    ELSIF (_eJobReslt = E_PROGRESS.PROGRESS_DONE)
    THEN
      _eState                   := E_PROGRESS.PROGRESS_CHECK;
      _eJobReslt                := _GroupItf.Enable(FALSE);
    END_IF
END_CASE
//-----------------------------------------------------------------------------
//-----------------------------------------------------------------------------
CASE _eState
OF
  E_PROGRESS.PROGRESS_CHECK:
    IF (_GroupInfo.GroupStandby) OR
       (_GroupInfo.GroupMoving)  OR
       (_GroupInfo.GroupNotReady)
    THEN
      _eState                   := E_PROGRESS.PROGRESS_DONE;

      IF (_eMessageLevel = E_MessageType.eMessageVerbose)
      THEN
        _stMsg.eType            := E_MessageType.eMessageVerbose;
        _stMsg.eSubdevice       := e_Subdevice.TransportUnit_General;
        _stMsg.iErrorNumber     := 0;
        _stMsg.sText            := concat( 'State: ', TO_STRING(THIS^._eState));
        _stMsg.sText            := concat(_stMsg.sText, ': ');
        _stMsg.sText            := concat(_stMsg.sText, TO_STRING(_eState));
        f_MessageSet(_stMsg, _nXpu);
      END_IF
    ELSE
      IF (_GroupInfo.GroupErrorStop) OR
         (_GroupInfo.GroupError)
      THEN
        _eState                 := E_PROGRESS.PROGRESS_ERROR;
      END_IF
    END_IF
END_CASE
//-----------------------------------------------------------------------------
//-----------------------------------------------------------------------------
GroupEnable                     := _eState;
END_METHOD

PROPERTY GroupInfo : REFERENCE TO ST_GROUP_INFO
SET
_GroupInfo REF= GroupInfo;
END_SET
END_PROPERTY

PROPERTY GroupItf : I_XtsTransport_CaGroup
SET
_GroupItf := GroupItf;
END_SET
END_PROPERTY

METHOD GroupStop : E_PROGRESS
VAR_INPUT
  Execute     : BOOL;
END_VAR
VAR_INST
  _nRepeat,
  _nStation,
  _nErrorId   : UDINT;
  _eJobReslt,
  _eState     : E_PROGRESS;
END_VAR
//-----------------------------------------------------------------------------
IF NOT Execute 
THEN 
	_eState                      := E_PROGRESS.PROGRESS_INIT; 
END_IF 
//-----------------------------------------------------------------------------
IF NOT Check() 
THEN 
	GroupStop                    := E_PROGRESS.PROGRESS_ERROR; 
	RETURN; 
END_IF
//-----------------------------------------------------------------------------
//-----------------------------------------------------------------------------
CASE _eState
OF
  E_PROGRESS.PROGRESS_INIT:
    IF Execute
    THEN
      _nRepeat                  :=
      _nErrorId                 := 0;
      _eJobReslt                := _GroupItf.Stop(FALSE);

      _eState                   := E_PROGRESS.PROGRESS_BUSY;
    END_IF
END_CASE
//---------------------------------------------------------------------------
//---------------------------------------------------------------------------
CASE _eState
OF
  E_PROGRESS.PROGRESS_BUSY:
    _eJobReslt                  := _GroupItf.Stop(TRUE);

    IF (_eJobReslt = E_PROGRESS.PROGRESS_ERROR)
    THEN
      _eState                   := E_PROGRESS.PROGRESS_PREPARE;
      _nErrorId                 := _GroupInfo.GroupErrorId;
      _eJobReslt                := _GroupItf.Stop(FALSE);

    ELSIF (_eJobReslt = E_PROGRESS.PROGRESS_DONE)
    THEN
      _eState                   := E_PROGRESS.PROGRESS_WORKING;
      _eJobReslt                := _GroupItf.Stop(FALSE);
    END_IF
END_CASE
//-----------------------------------------------------------------------------
//-----------------------------------------------------------------------------
CASE _eState
OF
  E_PROGRESS.PROGRESS_WORKING:
    IF NOT (_GroupInfo.GroupError)
    THEN
      _eState                   := E_PROGRESS.PROGRESS_DONE;

      IF (_eMessageLevel = E_MessageType.eMessageVerbose)
      THEN
        _stMsg.eType            := E_MessageType.eMessageVerbose;
        _stMsg.eSubdevice       := e_Subdevice.TransportUnit_General;
        _stMsg.iErrorNumber     := 0;
        _stMsg.sText            := concat( 'State: ', TO_STRING(THIS^._eState));
        _stMsg.sText            := concat(_stMsg.sText, ': ');
        _stMsg.sText            := concat(_stMsg.sText, TO_STRING(_eState));
        f_MessageSet(_stMsg, _nXpu);
      END_IF
    ELSE
      IF (_GroupInfo.GroupErrorStop) OR
         (_GroupInfo.GroupError)
      THEN
        _nRepeat                := _nRepeat + 1;
        IF NOT (_nRepeat > 2)
        THEN
          _eState               := E_PROGRESS.PROGRESS_BUSY;
        ELSE
          _eState               := E_PROGRESS.PROGRESS_ERROR;
        END_IF
      END_IF
    END_IF
END_CASE
//-----------------------------------------------------------------------------
//-----------------------------------------------------------------------------

GroupStop                       := _eState;
END_METHOD

PROPERTY MessageLevel : e_messagetype
SET
_eMessageLevel := MessageLevel;
END_SET
END_PROPERTY

METHOD MoverDisableAll : e_progress
VAR_INPUT
  Execute     : BOOL;
END_VAR
VAR_INST
  _nMover     : UINT;
  _nErrorId   : UDINT;
  _eRslt,
  _eState     : E_PROGRESS;
END_VAR
//-----------------------------------------------------------------------------
IF NOT Execute 
THEN 
	_eState                       := E_PROGRESS.PROGRESS_INIT; 
END_IF 
//-----------------------------------------------------------------------------
IF NOT Check() 
THEN 
	MoverDisableAll               := E_PROGRESS.PROGRESS_ERROR; 
	RETURN; 
END_IF
//-----------------------------------------------------------------------------
//-----------------------------------------------------------------------------
CASE _eState
OF
  E_PROGRESS.PROGRESS_INIT:
    IF Execute
    THEN
      _nErrorId                 := 0;
      _nMover                   := 1;

      _eState                   := E_PROGRESS.PROGRESS_BUSY;
    END_IF
END_CASE
//-----------------------------------------------------------------------------
//-----------------------------------------------------------------------------
CASE _eState
OF
  E_PROGRESS.PROGRESS_BUSY:
    _eState                     := E_PROGRESS.PROGRESS_PREPARE;
    _eRslt                      := _MoverItf[_nMover].Disable(FALSE);
    _eRslt                      := _MoverItf[_nMover].Reset(FALSE);
END_CASE
//-----------------------------------------------------------------------------
//-----------------------------------------------------------------------------
CASE _eState
OF
  E_PROGRESS.PROGRESS_PREPARE:
    _eRslt                      := _MoverItf[_nMover].Disable(TRUE);

    IF (_eRslt = E_PROGRESS.PROGRESS_ERROR)
    THEN
      _eState                   := E_PROGRESS.PROGRESS_BUSY;
      _nErrorId                 := _MoverInfo[_nMover].nErrorId; 
      _eRslt                    := _MoverItf[_nMover].Disable(FALSE);
      _MoverItf[_nMover].Reset(TRUE);

    ELSIF (_eRslt = E_PROGRESS.PROGRESS_DONE)
    THEN
      _eState                   := E_PROGRESS.PROGRESS_STARTUP;
    END_IF
END_CASE
//-----------------------------------------------------------------------------
//-----------------------------------------------------------------------------
CASE _eState
OF
  E_PROGRESS.PROGRESS_STARTUP:
    _eState                     := E_PROGRESS.PROGRESS_CHECK;
    _eRslt                      := _MoverItf[_nMover].Disable(FALSE);
END_CASE
//-----------------------------------------------------------------------------
//-----------------------------------------------------------------------------
CASE _eState
OF
  E_PROGRESS.PROGRESS_CHECK:
    IF (_nMover > MAX_MOVER-1)
    THEN
      _eState                   := E_PROGRESS.PROGRESS_DONE;

      IF (_eMessageLevel = E_MessageType.eMessageVerbose)
      THEN
        _stMsg.eType            := E_MessageType.eMessageVerbose;
        _stMsg.eSubdevice       := e_Subdevice.TransportUnit_General;
        _stMsg.iErrorNumber     := 0;
        _stMsg.sText            := concat( 'State: ', TO_STRING(THIS^._eState));
        _stMsg.sText            := concat(_stMsg.sText, ': ');
        _stMsg.sText            := concat(_stMsg.sText, TO_STRING(_eState));
        f_MessageSet(_stMsg, _nXpu);
      END_IF
    ELSE
      _nMover                   := _nMover + 1;
      _eState                   := E_PROGRESS.PROGRESS_BUSY;
    END_IF
END_CASE
//-----------------------------------------------------------------------------
//-----------------------------------------------------------------------------

MoverDisableAll                 := _eState;
END_METHOD

METHOD MoverEnableAll : e_progress
VAR_INPUT
  Execute     : BOOL;
END_VAR
VAR_INST
  _nMover     : UINT;
  _nErrorId   : UDINT;
  _eRslt,
  _eState     : E_PROGRESS;
END_VAR
//-----------------------------------------------------------------------------
IF NOT Execute 
THEN 
	_eState                       := E_PROGRESS.PROGRESS_INIT; 
END_IF 
//-----------------------------------------------------------------------------
IF NOT Check() 
THEN 
	MoverEnableAll                := E_PROGRESS.PROGRESS_ERROR; 
	RETURN; 
END_IF
//-----------------------------------------------------------------------------
//-----------------------------------------------------------------------------
CASE _eState
OF
  E_PROGRESS.PROGRESS_INIT:
    IF Execute
    THEN
      _nErrorId                 := 0;
      _nMover                   := 1;

      _eState                   := E_PROGRESS.PROGRESS_BUSY;
    END_IF
END_CASE
//-----------------------------------------------------------------------------
//-----------------------------------------------------------------------------
CASE _eState
OF
  E_PROGRESS.PROGRESS_BUSY:
    _eState                     := E_PROGRESS.PROGRESS_PREPARE;
    _eRslt                      := _MoverItf[_nMover].Enable(FALSE);
    _eRslt                      := _MoverItf[_nMover].Reset (FALSE);
END_CASE
//-----------------------------------------------------------------------------
//-----------------------------------------------------------------------------
CASE _eState
OF
  E_PROGRESS.PROGRESS_PREPARE:
    _eRslt                      := _MoverItf[_nMover].Enable(TRUE);

    IF (_eRslt = E_PROGRESS.PROGRESS_ERROR)
    THEN
      _eState                   := E_PROGRESS.PROGRESS_BUSY;
      _nErrorId                 := _MoverInfo[_nMover].nErrorId;
      _MoverItf[_nMover].Reset (TRUE);

    ELSIF (_eRslt = E_PROGRESS.PROGRESS_DONE)
    THEN
      _eState                   := E_PROGRESS.PROGRESS_STARTUP;
    END_IF
END_CASE
//-----------------------------------------------------------------------------
//-----------------------------------------------------------------------------
CASE _eState
OF
  E_PROGRESS.PROGRESS_STARTUP:
    _eState                     := E_PROGRESS.PROGRESS_CHECK;
    _eRslt                      := _MoverItf[_nMover].Enable(FALSE);
END_CASE
//-----------------------------------------------------------------------------
//-----------------------------------------------------------------------------
CASE _eState
OF
  E_PROGRESS.PROGRESS_CHECK:
    IF (_nMover > MAX_MOVER-1)
    THEN
      _eState                   := E_PROGRESS.PROGRESS_DONE;
      IF (_eMessageLevel = E_MessageType.eMessageVerbose)
      THEN
        _stMsg.eType            := E_MessageType.eMessageVerbose;
        _stMsg.eSubdevice       := e_Subdevice.TransportUnit_General;
        _stMsg.iErrorNumber     := 0;
        _stMsg.sText            := concat( 'State: ', TO_STRING(THIS^._eState));
        _stMsg.sText            := concat(_stMsg.sText, ': ');
        _stMsg.sText            := concat(_stMsg.sText, TO_STRING(_eState));
        f_MessageSet(_stMsg, _nXpu);
      END_IF
    ELSE
      _nMover                   := _nMover + 1;
      _eState                   := E_PROGRESS.PROGRESS_BUSY;
    END_IF
END_CASE
//-----------------------------------------------------------------------------
//-----------------------------------------------------------------------------

MoverEnableAll                  := _eState;
END_METHOD

METHOD MoverHaltAll : e_progress
VAR_INPUT
  Execute     : BOOL;
END_VAR
VAR_INST
  _nMover     : UINT;
  _nErrorId   : UDINT;
  _eRslt,
  _eState     : E_PROGRESS;
  _stMoveData : ST_MOVE_DATA; // dyn constraints for _MoverItf[i].Halt(Execute, stMoveData)
END_VAR
//-----------------------------------------------------------------------------
IF NOT Execute 
THEN 
	_eState                       := E_PROGRESS.PROGRESS_INIT; 
END_IF 
//-----------------------------------------------------------------------------
IF NOT Check() 
THEN 
	MoverHaltAll                  := E_PROGRESS.PROGRESS_ERROR; 
	RETURN; 
END_IF
//-----------------------------------------------------------------------------
//-----------------------------------------------------------------------------
CASE _eState
OF
  E_PROGRESS.PROGRESS_INIT:
    IF Execute
    THEN
      _nErrorId                 := 0;
      _nMover                   := 1;

      _eState                   := E_PROGRESS.PROGRESS_BUSY;
    END_IF
END_CASE
//-----------------------------------------------------------------------------
//-----------------------------------------------------------------------------
CASE _eState
OF
  E_PROGRESS.PROGRESS_BUSY:
    _eState                     := E_PROGRESS.PROGRESS_PREPARE;
    _stMoveData.rAcc            := _StationStart.rAccDec;
    _stMoveData.rGap            := _MoverLastGap[_nMover];

    IF NOT (_GroupInfo.AxisCount = MAX_MOVER)
    THEN
      _eRslt                    := _MoverItf[_nMover].Halt(FALSE, _stMoveData);
    ELSE
      _eRslt                    := _MoverItf[_nMover].HaltCa(FALSE, _stMoveData);
    END_IF
END_CASE
//-----------------------------------------------------------------------------
//-----------------------------------------------------------------------------
CASE _eState
OF
  E_PROGRESS.PROGRESS_PREPARE:
    IF NOT (_GroupInfo.AxisCount = MAX_MOVER)
    THEN
      _eRslt                    := _MoverItf[_nMover].Halt(TRUE, _stMoveData);
    ELSE
      _eRslt                    := _MoverItf[_nMover].HaltCa(TRUE, _stMoveData);
    END_IF

    IF (_eRslt = E_PROGRESS.PROGRESS_ERROR)
    THEN
      _eState                   := E_PROGRESS.PROGRESS_WORKING; // reset error on purpose, since we have to come back and get everybody in standstill
      _eRslt                    := _MoverItf[_nMover].Reset(FALSE);
      _nErrorId                 := _MoverInfo[_nMover].nErrorId; 

    ELSIF (_eRslt = E_PROGRESS.PROGRESS_DONE)
    THEN
      _eState                   := E_PROGRESS.PROGRESS_STARTUP;
    END_IF
END_CASE
//-----------------------------------------------------------------------------
//-----------------------------------------------------------------------------
CASE _eState
OF
  E_PROGRESS.PROGRESS_STARTUP:
    _eState                     := E_PROGRESS.PROGRESS_CHECK;

    IF NOT (_GroupInfo.AxisCount = MAX_MOVER)
    THEN
      _eRslt                    := _MoverItf[_nMover].Halt(FALSE, _stMoveData);
    ELSE
      _eRslt                    := _MoverItf[_nMover].HaltCa(FALSE, _stMoveData);
    END_IF

END_CASE
//-----------------------------------------------------------------------------
//-----------------------------------------------------------------------------
CASE _eState
OF
  E_PROGRESS.PROGRESS_CHECK:
    IF (_nMover > MAX_MOVER-1)
    THEN
      _eState                   := E_PROGRESS.PROGRESS_OCCUPIED;
    ELSE
      _nMover                   := _nMover + 1;
      _eState                   := E_PROGRESS.PROGRESS_BUSY;
    END_IF
END_CASE
//-----------------------------------------------------------------------------
//-----------------------------------------------------------------------------
CASE _eState
OF
  E_PROGRESS.PROGRESS_OCCUPIED:
    IF (_GroupInfo.AllAxesStanding)
    THEN
      _eState                   := E_PROGRESS.PROGRESS_DONE;

      IF (_eMessageLevel = E_MessageType.eMessageVerbose)
      THEN
        _stMsg.eType            := E_MessageType.eMessageVerbose;
        _stMsg.eSubdevice       := e_Subdevice.TransportUnit_General;
        _stMsg.iErrorNumber     := 0;
        _stMsg.sText            := concat( 'State: ', TO_STRING(THIS^._eState));
        _stMsg.sText            := concat(_stMsg.sText, ': ');
        _stMsg.sText            := concat(_stMsg.sText, TO_STRING(_eState));
        f_MessageSet(_stMsg, _nXpu);
      END_IF
    ELSE
      _nMover                   := 1;
      _eState                   := E_PROGRESS.PROGRESS_BUSY;
    END_IF
END_CASE
//-----------------------------------------------------------------------------
//-----------------------------------------------------------------------------
CASE _eState
OF
  E_PROGRESS.PROGRESS_WORKING:
    _eRslt                      := _MoverItf[_nMover].Reset(TRUE);

    IF (_eRslt = E_PROGRESS.PROGRESS_ERROR)
    THEN
      _eRslt                    := _MoverItf[_nMover].Reset(FALSE);
      _nErrorId                 := _MoverInfo[_nMover].nErrorId; 

    ELSIF (_eRslt = E_PROGRESS.PROGRESS_DONE)
    THEN
      _eState                   := E_PROGRESS.PROGRESS_BUSY;
      _eRslt                    := _MoverItf[_nMover].Reset(FALSE);
    END_IF
END_CASE
//-----------------------------------------------------------------------------
//-----------------------------------------------------------------------------

MoverHaltAll                    := _eState;
END_METHOD

PROPERTY MoverInfo : REFERENCE TO ARRAY[1..MAX_MOVER] OF ST_MOVER_INFO
SET
_MoverInfo REF= MoverInfo;
END_SET
END_PROPERTY

PROPERTY MoverItf : reference TO ARRAY[1..MAX_MOVER] OF I_XtsTransport_Mover
SET
_MoverItf REF= MoverItf;
END_SET
END_PROPERTY

PROPERTY MoverLastGap : REFERENCE to ARRAY[1..MAX_MOVER] of LREAL
SET
_MoverLastGap REF= MoverLastGap;
END_SET
END_PROPERTY

PROPERTY MoverLastPosition : REFERENCE to ARRAY[1..MAX_MOVER] of LREAL
SET
_MoverLastPosition REF= MoverLastPosition;
END_SET
END_PROPERTY

METHOD MoverStopAll : e_progress
VAR_INPUT
  Execute     : BOOL;
END_VAR
VAR_INST
  _nMover     : UINT;
  _nErrorId   : UDINT;
  _eRslt,
  _eState     : E_PROGRESS;
  _stMoveData : ST_MOVE_DATA; // dyn constraints for _MoverItf[i].Halt(Execute, stMoveData)
END_VAR
//-----------------------------------------------------------------------------
IF NOT Execute 
THEN 
	_eState                       := E_PROGRESS.PROGRESS_INIT; 
END_IF 
//-----------------------------------------------------------------------------
IF NOT Check() 
THEN 
	MoverStopAll                  := E_PROGRESS.PROGRESS_ERROR; 
	RETURN; 
END_IF
//-----------------------------------------------------------------------------
//-----------------------------------------------------------------------------
CASE _eState
OF
  E_PROGRESS.PROGRESS_INIT:
    IF Execute
    THEN
      _nErrorId                 := 0;
      _nMover                   := 1;

      _eState                   := E_PROGRESS.PROGRESS_BUSY;
    END_IF
END_CASE
//-----------------------------------------------------------------------------
//-----------------------------------------------------------------------------
CASE _eState
OF
  E_PROGRESS.PROGRESS_BUSY:
    _eState                     := E_PROGRESS.PROGRESS_PREPARE;
    _stMoveData.rAcc            := _StationStart.rAccDec;
    _stMoveData.rGap            := _MoverLastGap[_nMover];

    _eRslt                      := _MoverItf[_nMover].Stop(FALSE, _stMoveData);
END_CASE
//-----------------------------------------------------------------------------
//-----------------------------------------------------------------------------
CASE _eState
OF
  E_PROGRESS.PROGRESS_PREPARE:
    _eRslt                      := _MoverItf[_nMover].Stop(TRUE, _stMoveData);

    IF (_eRslt = E_PROGRESS.PROGRESS_ERROR)
    THEN
      _eState                   := E_PROGRESS.PROGRESS_WORKING; // reset error on purpose, since we have to come back and get everybody in standstill
      _eRslt                    := _MoverItf[_nMover].Reset(FALSE);
      _nErrorId                 := _MoverInfo[_nMover].nErrorId; 

    ELSIF (_eRslt = E_PROGRESS.PROGRESS_DONE)
    THEN
      _eState                   := E_PROGRESS.PROGRESS_STARTUP;
    END_IF
END_CASE
//-----------------------------------------------------------------------------
//-----------------------------------------------------------------------------
CASE _eState
OF
  E_PROGRESS.PROGRESS_STARTUP:
    _eState                     := E_PROGRESS.PROGRESS_CHECK;
    _eRslt                      := _MoverItf[_nMover].Halt(FALSE, _stMoveData);
END_CASE
//-----------------------------------------------------------------------------
//-----------------------------------------------------------------------------
CASE _eState
OF
  E_PROGRESS.PROGRESS_CHECK:
    IF (_nMover > MAX_MOVER-1)
    THEN
      _eState                   := E_PROGRESS.PROGRESS_OCCUPIED;
    ELSE
      _nMover                   := _nMover + 1;
      _eState                   := E_PROGRESS.PROGRESS_BUSY;
    END_IF
END_CASE
//-----------------------------------------------------------------------------
//-----------------------------------------------------------------------------
CASE _eState
OF
  E_PROGRESS.PROGRESS_OCCUPIED:
    IF (_GroupInfo.AllAxesStanding)
    THEN
      _eState                   := E_PROGRESS.PROGRESS_DONE;

      IF (_eMessageLevel = E_MessageType.eMessageVerbose)
      THEN
        _stMsg.eType            := E_MessageType.eMessageVerbose;
        _stMsg.eSubdevice       := e_Subdevice.TransportUnit_General;
        _stMsg.iErrorNumber     := 0;
        _stMsg.sText            := concat( 'State: ', TO_STRING(THIS^._eState));
        _stMsg.sText            := concat(_stMsg.sText, ': ');
        _stMsg.sText            := concat(_stMsg.sText, TO_STRING(_eState));
        f_MessageSet(_stMsg, _nXpu);
      END_IF
    ELSE
      _nMover                   := 1;
      _eState                   := E_PROGRESS.PROGRESS_BUSY;
    END_IF
END_CASE
//-----------------------------------------------------------------------------
//-----------------------------------------------------------------------------
CASE _eState
OF
  E_PROGRESS.PROGRESS_WORKING:
    _eRslt                      := _MoverItf[_nMover].Reset(TRUE);

    IF (_eRslt = E_PROGRESS.PROGRESS_ERROR)
    THEN
      _eRslt                    := _MoverItf[_nMover].Reset(FALSE);
      _nErrorId                 := _MoverInfo[_nMover].nErrorId; 

    ELSIF (_eRslt = E_PROGRESS.PROGRESS_DONE)
    THEN
      _eState                   := E_PROGRESS.PROGRESS_BUSY;
      _eRslt                    := _MoverItf[_nMover].Reset(FALSE);
    END_IF
END_CASE
//-----------------------------------------------------------------------------
//-----------------------------------------------------------------------------

MoverStopAll                    := _eState;
END_METHOD

PROPERTY State : REFERENCE TO ST_XTS_TRANSPORT_STATE
SET
_State ref= State;
END_SET
END_PROPERTY

PROPERTY StationControl : REFERENCE TO ARRAY[1..MAX_STATION]  OF ST_STATION_CTRL
SET
_StationControl REF= StationControl;
END_SET
END_PROPERTY

PROPERTY StationCtrlItf : REFERENCE TO ARRAY[1..MAX_STATION]  OF I_XtsTransport_Station;
SET
_ItfStationCtrl REF= StationCtrlItf;
END_SET
END_PROPERTY

PROPERTY StationListsItf : reference to ARRAY[1..MAX_STATION] OF I_Station_LinkedList
SET
_ItfStationList ref= StationListsItf;
END_SET
END_PROPERTY

METHOD StationsClearAll : E_PROGRESS
VAR_INPUT
  Execute     : BOOL;
END_VAR
VAR_INST
  _nStation,
  _nErrorId   : UDINT;
  _eJobReslt,
  _eState     : E_PROGRESS;
END_VAR
//-----------------------------------------------------------------------------
IF NOT Execute 
THEN 
	_eState                       := E_PROGRESS.PROGRESS_INIT; 
END_IF 
//-----------------------------------------------------------------------------
IF NOT Check() 
THEN 
	StationsClearAll              := E_PROGRESS.PROGRESS_ERROR; 
	RETURN; 
END_IF
//-----------------------------------------------------------------------------
//-----------------------------------------------------------------------------
CASE _eState
OF
  E_PROGRESS.PROGRESS_INIT:
    IF Execute
    THEN
      _nErrorId                 := 0;
      _nStation                 := 1;
      _eState                   := E_PROGRESS.PROGRESS_BUSY;
    END_IF
  //---------------------------------------------------------------------------
  //---------------------------------------------------------------------------
  E_PROGRESS.PROGRESS_BUSY:
    _eJobReslt                  := _ItfStationCtrl[_nStation].Init();

    IF (_eJobReslt = E_PROGRESS.PROGRESS_ERROR)
    THEN
      _eState                   := E_PROGRESS.PROGRESS_ERROR;
      _nErrorId                 := 669;

    ELSIF (_eJobReslt = E_PROGRESS.PROGRESS_DONE)
    THEN
      _eState                   := E_PROGRESS.PROGRESS_WORKING;
    END_IF

  //---------------------------------------------------------------------------
  //---------------------------------------------------------------------------
  E_PROGRESS.PROGRESS_WORKING:
    IF (_nStation < MAX_STATION)
    THEN
      _nStation                 := _nStation + 1;
      _eState                   := E_PROGRESS.PROGRESS_BUSY;
    ELSE
      _eState                   := E_PROGRESS.PROGRESS_DONE;

      IF (_eMessageLevel = E_MessageType.eMessageVerbose)
      THEN
        _stMsg.eType            := E_MessageType.eMessageVerbose;
        _stMsg.eSubdevice       := e_Subdevice.TransportUnit_General;
        _stMsg.iErrorNumber     := 0;
        _stMsg.sText            := concat( 'State: ', TO_STRING(THIS^._eState));
        _stMsg.sText            := concat(_stMsg.sText, ': ');
        _stMsg.sText            := concat(_stMsg.sText, TO_STRING(_eState));
        f_MessageSet(_stMsg, _nXpu);
      END_IF
    END_IF
END_CASE
//-----------------------------------------------------------------------------
//-----------------------------------------------------------------------------

StationsClearAll                := _eState;
END_METHOD

METHOD StationsClearOutfeed : e_progress
VAR_INPUT
  Execute         : BOOL;
END_VAR
VAR_INST
  _StnState       : ST_STATION_STATE;

  _nStation,
  _nMover         : UINT;

  _nErrorId       : UDINT;

  _eRslt,
  _eState         : E_PROGRESS;
  
  _stMsg          : ST_Message;
  _stMoveData     : ST_MOVE_DATA;
END_VAR
//-----------------------------------------------------------------------------
IF NOT Execute 
THEN 
	_eState                       := E_PROGRESS.PROGRESS_INIT; 
END_IF 
//-----------------------------------------------------------------------------
IF NOT Check() 
THEN 
	StationsClearOutfeed           := E_PROGRESS.PROGRESS_ERROR; 
	RETURN; 
END_IF
//-----------------------------------------------------------------------------
//-----------------------------------------------------------------------------
CASE _eState
OF
  E_PROGRESS.PROGRESS_INIT:
    IF Execute
    THEN
      _nErrorId                 := 0;

      _nStation                 :=
      _nMover                   := 1;

      _eState                   := E_PROGRESS.PROGRESS_BUSY;
    END_IF
END_CASE
//-----------------------------------------------------------------------------
//-----------------------------------------------------------------------------
CASE _eState
OF
  E_PROGRESS.PROGRESS_BUSY:
    _StnState                   := _StationState[_nStation];

    CASE _StnState.eState
    OF
      E_STATION_STATE.STATION_MOVER_RELEASE:
        _StationControl[_nStation].eCmd := E_STATION_CTRL.STATION_MOVER_GONE;

    ELSE
      _eState                   := E_PROGRESS.PROGRESS_PREPARE;  
    END_CASE
END_CASE
//-----------------------------------------------------------------------------
//-----------------------------------------------------------------------------
CASE _eState
OF
  E_PROGRESS.PROGRESS_PREPARE:
    IF (_nStation > MAX_STATION-1)
    THEN
      _eState                   := E_PROGRESS.PROGRESS_DONE;
    ELSE
      _nStation                 := _nStation + 1;
      _eState                   := E_PROGRESS.PROGRESS_BUSY;
    END_IF
END_CASE

StationsClearOutfeed             := _eState;
END_METHOD

PROPERTY StationStart : reference to ST_STATION_PARAMETER
SET
_StationStart REF= StationStart;
END_SET
END_PROPERTY

PROPERTY StationStartIndex : uint
GET
StationStartIndex := _nStartStation;
END_GET
SET
_nStartStation := StationStartIndex;
END_SET
END_PROPERTY

PROPERTY StationState : REFERENCE TO ARRAY[1..MAX_STATION]  OF ST_STATION_STATE
SET
_StationState REF= StationState;
END_SET
END_PROPERTY

METHOD Template : E_PROGRESS
VAR_INPUT
  Execute     : BOOL;
END_VAR
VAR_INST
  _nErrorId   : UDINT;
  _eState     : E_PROGRESS;
END_VAR
//-----------------------------------------------------------------------------
IF NOT Execute 
THEN 
	_eState                       := E_PROGRESS.PROGRESS_INIT; 
END_IF 
//-----------------------------------------------------------------------------
IF NOT Check() 
THEN 
	Template_1                    := E_PROGRESS.PROGRESS_ERROR; 
	RETURN; 
END_IF
//-----------------------------------------------------------------------------
//-----------------------------------------------------------------------------
CASE _eState
OF
  E_PROGRESS.PROGRESS_INIT:
    IF Execute
    THEN
      _nErrorId                 := 0;

      _eState                   := E_PROGRESS.PROGRESS_BUSY;
    END_IF
END_CASE
//-----------------------------------------------------------------------------
//-----------------------------------------------------------------------------
CASE _eState
OF
  E_PROGRESS.PROGRESS_BUSY:
    _eState                     := E_PROGRESS.PROGRESS_PREPARE;
END_CASE
//-----------------------------------------------------------------------------
//-----------------------------------------------------------------------------
CASE _eState
OF
  E_PROGRESS.PROGRESS_PREPARE:

    IF (.Error)
    THEN
      _eState                   := E_PROGRESS.PROGRESS_ERROR;
      _nErrorId                 := 


    ELSIF (.Done)
    THEN
      _eState                   := E_PROGRESS.;

    END_IF
END_CASE
//-----------------------------------------------------------------------------
//-----------------------------------------------------------------------------

Template_1                      := _eState;
END_METHOD

METHOD TransportRestart : e_progress // movers must already to be error free, enabled and added to CA Group
VAR_INPUT
  Execute         : BOOL;
END_VAR
VAR_INST
  _StnState       : ST_STATION_STATE;

  _nStation,
  _nMover         : UINT;

  _nErrorId       : UDINT;

  _eRslt,
  _eState         : E_PROGRESS;
  
  _stMsg          : ST_Message;
  _stMoveData     : ST_MOVE_DATA;
END_VAR
//-----------------------------------------------------------------------------
IF NOT Execute 
THEN 
	_eState                       := E_PROGRESS.PROGRESS_INIT; 
END_IF 
//-----------------------------------------------------------------------------
IF NOT Check() 
THEN 
	TransportRestart              := E_PROGRESS.PROGRESS_ERROR; 
	RETURN; 
END_IF
//-----------------------------------------------------------------------------
//-----------------------------------------------------------------------------
CASE _eState
OF
  E_PROGRESS.PROGRESS_INIT:
    IF Execute
    THEN
      _nErrorId                 := 0;

      _nStation                 :=
      _nMover                   := 1;

      IF (_GroupInfo.AxisCountEnabled = MAX_MOVER)
      THEN
        _eState                 := E_PROGRESS.PROGRESS_BUSY;
      ELSE
        _eState                 := E_PROGRESS.PROGRESS_ERROR;

        _stMsg.eType            := E_MessageType.eMessageError;
        _stMsg.eSubdevice       := e_Subdevice.TransportUnit_Restart;
        _stMsg.iErrorNumber     := _GroupInfo.AxisCountEnabled;
        _stMsg.sText            := TO_STRING(_eState);
        _stMsg.sText            := concat(_stMsg.sText, ': _GroupInfo.AxisCountEnabled <> MAX_MOVER');
        f_MessageSet(_stMsg, _nXpu);
      END_IF
    END_IF
END_CASE
//-----------------------------------------------------------------------------
//-----------------------------------------------------------------------------
CASE _eState
OF
  E_PROGRESS.PROGRESS_BUSY:
    _StnState                   := _StationState[_nStation];

    CASE _StnState.eState
    OF
      E_STATION_STATE.STATION_ERROR_INFEED_ERROR:
        _StationControl[_nStation].eCmd := E_STATION_CTRL.STATION_MOVER_ENTER_RETRY;

      E_STATION_STATE.STATION_ERROR_OUTFEED_ERROR:
        _StationControl[_nStation].eCmd := E_STATION_CTRL.STATION_MOVER_GONE;

      E_STATION_STATE.STATION_ERROR_FATAL:
        _eState                 := E_PROGRESS.PROGRESS_ERROR;

        _stMsg.eType            := E_MessageType.eMessageError;
        _stMsg.eSubdevice       := e_Subdevice.TransportUnit_Restart;
        _stMsg.iErrorNumber     := _nStation;
        _stMsg.sText            := TO_STRING(_eState);
        _stMsg.sText            := concat(_stMsg.sText, ': _nStation STATION_ERROR_FATAL');
        f_MessageSet(_stMsg, _nXpu);

    ELSE
      _eState                   := E_PROGRESS.PROGRESS_PREPARE;  
    END_CASE
END_CASE
//-----------------------------------------------------------------------------
//-----------------------------------------------------------------------------
CASE _eState
OF
  E_PROGRESS.PROGRESS_PREPARE:
    IF (_nStation > MAX_STATION-1)
    THEN
      _eState                   := E_PROGRESS.PROGRESS_STARTUP;
    ELSE
      _nStation                 := _nStation + 1;
      _eState                   := E_PROGRESS.PROGRESS_BUSY;
    END_IF
END_CASE
//-----------------------------------------------------------------------------
//-----------------------------------------------------------------------------
CASE _eState
OF
  E_PROGRESS.PROGRESS_STARTUP:
    _stMoveData.rPos            := _MoverLastPosition[_nMover];
    _stMoveData.rGap            := _MoverLastGap     [_nMover];

    _stMoveData.rVelo           := _StationStart.rVelo;
    _stMoveData.rAcc            := _StationStart.rAccDec;
    _stMoveData.rJerk           := _StationStart.rJerk;

    _stMoveData.rDelta          :=   0.1;
    _stMoveData.rDistance       :=  -1.0;
    _stMoveData.rOverride       := 100.0;

    _eRslt                      := _MoverItf[_nMover].SendToAbsPosCa(FALSE, _stMoveData);

    IF (_MoverInfo[_nMover].bMoverEnabled)
    THEN
      _eState                   := E_PROGRESS.PROGRESS_CHECK;
    END_IF
END_CASE
//-----------------------------------------------------------------------------
//-----------------------------------------------------------------------------
CASE _eState
OF
  E_PROGRESS.PROGRESS_CHECK:
    _eRslt                      := _MoverItf[_nMover].SendToAbsPosCa(TRUE, _stMoveData);

    IF (_eRslt = E_PROGRESS.PROGRESS_ERROR)
    THEN
      _eState                   := E_PROGRESS.PROGRESS_ERROR;

    ELSIF (_eRslt = E_PROGRESS.PROGRESS_DONE)
    THEN
      _eRslt                    := _MoverItf[_nMover].SendToAbsPosCa(FALSE, _stMoveData);
      _eState                   := E_PROGRESS.PROGRESS_OCCUPIED;
    END_IF
END_CASE
//-----------------------------------------------------------------------------
//-----------------------------------------------------------------------------
CASE _eState
OF
  E_PROGRESS.PROGRESS_OCCUPIED:
    IF (_nMover > MAX_MOVER-1)
    THEN
      _eState                   := E_PROGRESS.PROGRESS_DONE;

      IF (_eMessageLevel = E_MessageType.eMessageVerbose)
      THEN
        _stMsg.eType            := E_MessageType.eMessageVerbose;
        _stMsg.eSubdevice       := e_Subdevice.TransportUnit_General;
        _stMsg.iErrorNumber     := 0;
        _stMsg.sText            := concat( 'State: ', TO_STRING(THIS^._eState));
        _stMsg.sText            := concat(_stMsg.sText, ': ');
        _stMsg.sText            := concat(_stMsg.sText, TO_STRING(_eState));
        f_MessageSet(_stMsg, _nXpu);
      END_IF
    ELSE
      _nMover                   := _nMover + 1;
      _eState                   := E_PROGRESS.PROGRESS_STARTUP;
    END_IF
END_CASE
//-----------------------------------------------------------------------------
//-----------------------------------------------------------------------------

TransportRestart                := _eState;
END_METHOD

METHOD TransportStart : e_progress
VAR_INPUT
  Execute       : BOOL;
END_VAR
VAR_INST
  _nMover,
  _nStation     : UINT;
  _nErrorId     : UDINT;

  _stMoveData   : ST_MOVE_DATA;

  _eRslt,
  _eState       : E_PROGRESS;
  _stMsg        : ST_Message;
END_VAR
//-----------------------------------------------------------------------------
IF NOT Execute 
THEN 
	_eState                       := E_PROGRESS.PROGRESS_INIT; 
END_IF 
//-----------------------------------------------------------------------------
IF NOT Check() 
THEN 
	TransportStart                := E_PROGRESS.PROGRESS_ERROR; 
	RETURN; 
END_IF
//-----------------------------------------------------------------------------
//-----------------------------------------------------------------------------
CASE _eState
OF
  E_PROGRESS.PROGRESS_INIT:
    IF Execute
    THEN
      _nErrorId                 := 0;
      _nMover                   := 1;

      IF (_StationStart.rPosWait - (_MoverInfo[_nMover].rModuloActPos +0.1) < 0)
      THEN
        _stMoveData.rPos        := _StationStart.rPosWait + _MoverItf[_nMover].RailLength;
      ELSE
        _stMoveData.rPos        := _StationStart.rPosWait;
      END_IF

      _stMoveData.rGap          := _StationStart.rGap;

      _stMoveData.rVelo         := _StationStart.rVelo;
      _stMoveData.rAcc          := _StationStart.rAccDec;
      _stMoveData.rJerk         := _StationStart.rJerk;

      _stMoveData.rDelta        :=   0.05;
      _stMoveData.rDistance     :=  -1.0;     // distance used by SendToPosCa

      _stMoveData.rOverride     := 100.0;

      _eRslt                    := _MoverItf[_nMover].SendToModuloPosCa(FALSE, _stMoveData);
      _eRslt                    := _MoverItf[_nMover].SendToAbsPosCa(FALSE, _stMoveData);
      _eRslt                    := StationsClearAll(FALSE);

      IF (_GroupInfo.AxisCountEnabled = MAX_MOVER)
      THEN
        _eState                 := E_PROGRESS.PROGRESS_BUSY;
      ELSE
        _eState                 := E_PROGRESS.PROGRESS_ERROR;

        _stMsg.eType            := E_MessageType.eMessageError;
        _stMsg.eSubdevice       := e_Subdevice.TransportUnit_Start;
        _stMsg.iErrorNumber     := _GroupInfo.AxisCountEnabled;
        _stMsg.sText            := TO_STRING(_eState);
        _stMsg.sText            := concat(_stMsg.sText, ': _GroupInfo.AxisCountEnabled <> MAX_MOVER');
        f_MessageSet(_stMsg, _nXpu);
      END_IF
    END_IF

  //---------------------------------------------------------------------------
  E_PROGRESS.PROGRESS_BUSY:
    _eRslt                      := StationsClearAll(TRUE); // all xts station queues clear
    IF (_eRslt = E_PROGRESS.PROGRESS_DONE)
    THEN
      _eState                   := E_PROGRESS.PROGRESS_PREPARE;
    ELSE
      IF (_eRslt = E_PROGRESS.PROGRESS_ERROR)
      THEN
        _eState                 := E_PROGRESS.PROGRESS_ERROR;
      END_IF
    END_IF

  E_PROGRESS.PROGRESS_PREPARE:
    _eRslt                      := _MoverItf[_nMover].SendToModuloPosCa(TRUE, _stMoveData);

    IF (_eRslt = E_PROGRESS.PROGRESS_ERROR)
    THEN
      _eState                   := E_PROGRESS.PROGRESS_ERROR;
      _nErrorId                 := _MoverInfo[_nMover].nErrorId;
      _eRslt                    := _MoverItf[_nMover].SendToModuloPosCa(FALSE, _stMoveData); 

    ELSIF (_eRslt = E_PROGRESS.PROGRESS_DONE)
    THEN
      _eState                   := E_PROGRESS.PROGRESS_STARTUP;
      _eRslt                    := _MoverItf[_nMover].SendToModuloPosCa(FALSE, _stMoveData);
    END_IF

  //---------------------------------------------------------------------------
  E_PROGRESS.PROGRESS_STARTUP:
    IF (_nMover > MAX_MOVER-1)
    THEN
      // all mover are sent to start position, now prepare ticket for Mover 1
      _eState                         := E_PROGRESS.PROGRESS_CHECK;
      // ticket data
      _stMoverDataSend.nMask          := TO_USINT(EXPT(2,_StationStart.nConfiguredStopCount))-1;
      _stMoverDataSend.nMoverId       := TO_USINT(1);
      _stMoverDataSend.nTargetStation := TO_USINT(_nStartStation);
  
      IF (_nStartStation > 0) AND
         (_nStartStation < MAX_STATION+1)
      THEN
        _stListResult           := _ItfStationList[_nStartStation].AddTailValue(_stMoverDataSend); // add first mover to list of _ItfStations[_nStartStation]
      END_IF

    ELSE
      _nMover                   := _nMover + 1;                                                 // increment mover ID
      _stMoveData.rPos          := _StationStart.rPosWait + 2*_MoverItf[_nMover].RailLength;    // all other mover are commanded an extra round, to make sure that mover 1 is always leading the pack
      _eRslt                    := _MoverItf[_nMover].SendToModuloPosCa(FALSE, _stMoveData);
      _eRslt                    := _MoverItf[_nMover].SendToAbsPosCa(FALSE, _stMoveData);
      _eState                   := E_PROGRESS.PROGRESS_PREPARE;                                 // go back and trigger move
    END_IF

  //---------------------------------------------------------------------------
  E_PROGRESS.PROGRESS_CHECK:
    IF (_MoverInfo[1].bMoverInTarget)
    THEN
      IF (_GroupInfo.AllAxesStanding) // wait for all mover standstill
      THEN
        _stMoveData.rPos        := _MoverInfo[1].rAbsTargetPos;                    // Mover1 position to retrigger the movers

        IF (MAX_MOVER > 1)
        THEN
          _nMover               := 2;
          IF (_stMoveData.rPos < _MoverInfo[_nMover].rAbsActPos)
          THEN
            _stMoveData.rPos    := _stMoveData.rPos + _MoverItf[_nMover].RailLength;
          END_IF
          _eState               := E_PROGRESS.PROGRESS_OCCUPIED;
        ELSE
          _eState               := E_PROGRESS.PROGRESS_WORKING;
        END_IF
      END_IF
    END_IF

  //---------------------------------------------------------------------------
  E_PROGRESS.PROGRESS_OCCUPIED:
    _eRslt                      := _MoverItf[_nMover].SendToAbsPosCa(TRUE, _stMoveData); // retrigger

    IF (_eRslt = E_PROGRESS.PROGRESS_ERROR)
    THEN
      _eState                   := E_PROGRESS.PROGRESS_ERROR;
      _nErrorId                 := _MoverInfo[_nMover].nErrorId;
      _eRslt                    := _MoverItf[_nMover].SendToAbsPosCa(FALSE, _stMoveData); 

    ELSIF (_eRslt = E_PROGRESS.PROGRESS_DONE)
    THEN
      _eState                   := E_PROGRESS.PROGRESS_WORKING;
      _eRslt                    := _MoverItf[_nMover].SendToAbsPosCa(FALSE, _stMoveData);

      // write ticket for mover in station list
      _stMoverDataSend.nMask          := TO_USINT(EXPT(2,_StationStart.nConfiguredStopCount))-1;
      _stMoverDataSend.nMoverId       := TO_USINT(_nMover);
      _stMoverDataSend.nTargetStation := TO_USINT(_nStartStation);

      IF (_nStartStation > 0) AND
         (_nStartStation < MAX_STATION+1)
      THEN
        _stListResult                 := _ItfStationList[_nStartStation].AddTailValue(_stMoverDataSend); // enter in list
      END_IF
    END_IF

  //---------------------------------------------------------------------------
  E_PROGRESS.PROGRESS_WORKING:
    IF (_nMover > MAX_MOVER-1)
    THEN
      _eState                   := E_PROGRESS.PROGRESS_DONE;

      IF (_eMessageLevel = E_MessageType.eMessageVerbose)
      THEN
        _stMsg.eType            := E_MessageType.eMessageVerbose;
        _stMsg.eSubdevice       := e_Subdevice.TransportUnit_General;
        _stMsg.iErrorNumber     := 0;
        _stMsg.sText            := concat( 'State: ', TO_STRING(THIS^._eState));
        _stMsg.sText            := concat(_stMsg.sText, ': ');
        _stMsg.sText            := concat(_stMsg.sText, TO_STRING(_eState));
        f_MessageSet(_stMsg, _nXpu);
      END_IF
    ELSE
      _nMover                   := _nMover + 1;
      IF (_stMoveData.rPos < _MoverInfo[_nMover].rAbsActPos)
      THEN
        _stMoveData.rPos        := _stMoveData.rPos + _MoverItf[_nMover].RailLength;
      END_IF
      _eState                   := E_PROGRESS.PROGRESS_OCCUPIED;
    END_IF
END_CASE
//-----------------------------------------------------------------------------
//-----------------------------------------------------------------------------

TransportStart                  := _eState;
END_METHOD

PROPERTY XpuCtrl : REFERENCE TO ST_XPU_CTRL
SET
_XpuCtrl REF= XpuCtrl;
END_SET
END_PROPERTY

PROPERTY XpuInfo : REFERENCE TO ST_XPU_INFO
SET
_XpuInfo REF= XpuInfo;
END_SET
END_PROPERTY

METHOD XpuInit : E_PROGRESS
VAR_INPUT
  Execute     : BOOL;
END_VAR
VAR_INST
  _nErrorId   : UDINT;
  _eJobReslt,
  _eState     : E_PROGRESS;
END_VAR
//-----------------------------------------------------------------------------
IF NOT Execute 
THEN 
	_eState                       := E_PROGRESS.PROGRESS_INIT; 
END_IF 
//-----------------------------------------------------------------------------
IF NOT Check() 
THEN 
	XpuInit                       := E_PROGRESS.PROGRESS_ERROR; 
	RETURN; 
END_IF
//-----------------------------------------------------------------------------
//-----------------------------------------------------------------------------
CASE _eState
OF
  E_PROGRESS.PROGRESS_INIT:
    IF Execute
    THEN
      _nErrorId                 := 0;
      _XpuCtrl.Cmd              := E_XPU_CTRL.XTS_CMD_NULL; // clear interface

      _eState                   := E_PROGRESS.PROGRESS_BUSY;
    END_IF
  //---------------------------------------------------------------------------
  //---------------------------------------------------------------------------
  E_PROGRESS.PROGRESS_BUSY:
    _XpuCtrl.Cmd                := E_XPU_CTRL.XTS_CMD_INIT; // start Xpu init

    IF (f_GetProgress(_XpuState.State) = E_PROGRESS.PROGRESS_DONE)         // check Xpu init done
    THEN
      _eState                   := E_PROGRESS.PROGRESS_PREPARE;

    ELSIF (f_GetProgress(_XpuState.State) = E_PROGRESS.PROGRESS_ERROR)     // check for error
    THEN
      _eState                   := E_PROGRESS.PROGRESS_ERROR;
    END_IF
  //---------------------------------------------------------------------------
  //---------------------------------------------------------------------------
  E_PROGRESS.PROGRESS_PREPARE:
    _XpuCtrl.Cmd                := E_XPU_CTRL.XTS_IDLE;     // Xpu start cyclic checks and mover detection

    IF (f_GetProgress(_XpuState.State) = E_PROGRESS.PROGRESS_ERROR)     // check for error
    THEN
      _eState                   := E_PROGRESS.PROGRESS_ERROR;

    ELSIF (f_GetProgress(_XpuState.State) = E_PROGRESS.PROGRESS_WORKING)      // check Xpu Idle working
    THEN
      _eState                   := E_PROGRESS.PROGRESS_STARTUP;

    END_IF
  //---------------------------------------------------------------------------
  //---------------------------------------------------------------------------
  E_PROGRESS.PROGRESS_STARTUP:
    IF (f_GetProgress(_XpuState.State) = E_PROGRESS.PROGRESS_ERROR)
    THEN
      _eState                   := E_PROGRESS.PROGRESS_ERROR;

    ELSIF (_XpuState.Check = E_XPU_CHECK.MOVER_ID_SIMULATION) OR
          (_XpuState.Check = E_XPU_CHECK.MOVER_ID_STANDARD)   OR
          (_XpuState.Check = E_XPU_CHECK.MOVER_ID_DETECTION_VALID)
    THEN
      _eState                   := E_PROGRESS.PROGRESS_DONE;

      IF (_eMessageLevel = E_MessageType.eMessageVerbose)
      THEN
        _stMsg.eType            := E_MessageType.eMessageVerbose;
        _stMsg.eSubdevice       := e_Subdevice.TransportUnit_General;
        _stMsg.iErrorNumber     := 0;
        _stMsg.sText            := concat( 'State: ', TO_STRING(THIS^._eState));
        _stMsg.sText            := concat(_stMsg.sText, ': ');
        _stMsg.sText            := concat(_stMsg.sText, TO_STRING(_eState));
        f_MessageSet(_stMsg, _nXpu);
      END_IF
    END_IF
END_CASE
//-----------------------------------------------------------------------------
//-----------------------------------------------------------------------------
XpuInit                         := _eState;
END_METHOD

PROPERTY XpuInstance : uint
SET
//
// Who am I?
// Environment may have more than one ProcessingUnit,
// information required for connecting to the correct instance of ProcessingUnit
_nXpu := XpuInstance;
END_SET
END_PROPERTY

PROPERTY XpuState : REFERENCE TO ST_XPU_STATE
SET
_XpuState ref= XpuState;
END_SET
END_PROPERTY

END_FUNCTION_BLOCK

// ---- XTS/Xpu/fb_XpuCtrl.TcPOU
//---------------------------------------------------------------------------------------------------------------
//
//  HAUD 2023.12.15
//
//  - XTS_TRANSPORT_LAYER
//
//  - fb_XpuCtrl extends fb_Xpu
//  CTRL / STATE --> see proprerties
//  structs for use of function block via mapping
//  cyclic check for new command
//
//  VAR INPUT / OUTPUT --> see properties
//
//---------------------------------------------------------------------------------------------------------------
// This SOFTWARE is provided as an Exemple by THE PROVIDER "as is" and "with all faults." THE PROVIDER makes no 
// representations or warranties of any kind concerning the safety, suitability, lack of viruses, inaccuracies, 
// typographical errors, or other harmful components of this SOFTWARE. There are inherent dangers in the use of 
// any software, and you are solely responsible for determining whether this SOFTWARE is compatible with your 
// equipment and other software installed on your equipment. You are also solely responsible for the protection 
// of your equipment and backup of your data, and THE PROVIDER will not be liable for any damages you may suffer 
// in connection with using, modifying, or distributing this SOFTWARE.
//---------------------------------------------------------------------------------------------------------------
FUNCTION_BLOCK fb_XpuCtrl EXTENDS fb_Xpu
VAR
  _Ctrl                       : REFERENCE TO ST_XPU_CTRL;
  _State                      : REFERENCE TO ST_XPU_STATE;

  _eCmd,
  _eCmdOld                    : E_XPU_CTRL;

  _eResult                    : E_PROGRESS;
  _eState                     : E_XPU_STATE;

END_VAR

IF NOT Check() THEN RETURN; END_IF

_stMsg.eDevice                := e_Device.Xpu + _nXpu;

_eCmd                         := _Ctrl.Cmd;

// check for command change
// get state for cmd
IF (_eCmd <> _eCmdOld)
THEN
  _eState                     := Cmd(_eCmd);
  _eCmdOld                    := _eCmd;
END_IF


CASE _eState
OF
  E_XPU_STATE.XTS_INIT:       // get TcCOM information for connecting to XTS utility function blocks
    _eInit                    := XpuInit(TRUE, _eResult, _eCheck);
    _State.Check              := _eCheck;

  E_XPU_STATE.XTS_IDLE:       // cyclic check; add additional information if your application requires it
    _eResult                  := SUPER^.Cycle(TRUE, _eCheck);  // cyclic check of ProcessingUnit data

    IF NOT (_eResult = E_PROGRESS.PROGRESS_ERROR)
    THEN
      _State.Check            := DetectMoverId(TRUE); // mover detection is checked here
    ELSE
      _State.Check            := _eCheck;
    END_IF

ELSE
  _eResult                    := E_PROGRESS.PROGRESS_INVALID;
END_CASE


CASE _eResult
OF
  E_PROGRESS.PROGRESS_INVALID:
    _State.State              := TO_UINT(_eResult);

  E_PROGRESS.PROGRESS_ERROR:
    _State.State              := _eState + E_PROGRESS.PROGRESS_ERROR;

  E_PROGRESS.PROGRESS_DONE:
    _State.State              := _eState + E_PROGRESS.PROGRESS_DONE;

ELSE
  _State.State                := _eState + _eResult;
END_CASE

_State.Init                   := _eInit;
_State.DcLink                 := AllModulesDcLink;

METHOD Check : BOOL

IF NOT __ISVALIDREF(_Ctrl)
THEN
  _eCheck                     := E_XPU_CHECK.POINTER_NULL_CTRL;
  RETURN;
END_IF

IF NOT __ISVALIDREF(_State)
THEN
  _eCheck                     := E_XPU_CHECK.POINTER_NULL_STATE;
  RETURN;
END_IF

IF NOT (_nXpu <> 0)
THEN
  _eCheck                     := E_XPU_CHECK.XPU_INSTANCE_NULL;
  RETURN;
END_IF

Check                         := TRUE;
END_METHOD

METHOD PRIVATE Cmd : E_XPU_STATE
VAR_INPUT
  Ctrl      : E_XPU_CTRL;
END_VAR
VAR_INST
  _eState   : E_XPU_STATE;
  _eCk      : E_XPU_CHECK;
END_VAR
IF NOT Check() THEN RETURN; END_IF


CASE Ctrl
OF
  E_XPU_CTRL.XTS_CMD_NULL:  // clear all method calls
    _eState               := E_XPU_STATE.XTS_NULL;
    SUPER^.Cycle(FALSE, _eCk);
    DetectMoverId(FALSE);
    XpuInit(FALSE, _eResult, _eCheck);


  E_XPU_CTRL.XTS_CMD_INIT:  // clear methods for initialization
    _eState               := E_XPU_STATE.XTS_INIT;
    _eInit                := XpuInit(FALSE, _eResult, _eCheck);

ELSE
  IF NOT (_eInit = E_XPU_INIT.INIT_DONE)
  THEN
    // no init, no further commands possible
    _eState               := E_XPU_STATE.XTS_INVALID;
  ELSE
    CASE Ctrl
    OF
      E_XPU_CTRL.XTS_IDLE:  // clear methods for cyclic checks
        _eState           := E_XPU_STATE.XTS_IDLE;
        SUPER^.Cycle(FALSE, _eCk);
        DetectMoverId(FALSE);
    ELSE
        _eState           := E_XPU_STATE.XTS_INVALID;
    END_CASE
  END_IF
END_CASE

Cmd                       := _eState;
END_METHOD

PROPERTY Ctrl : REFERENCE TO ST_XPU_CTRL
SET
_Ctrl REF= Ctrl;
END_SET
END_PROPERTY

METHOD DetectMoverId  : E_XPU_CHECK
VAR_INPUT
  Enable                : BOOL;
END_VAR
VAR_INST
  _bInit                : BOOL;
  _eReturn,
  _eState               : E_XPU_CHECK;
  _nCheckModulo         : UINT := 500;
  _nCheckCount          : UINT;
END_VAR
//-----------------------------------------------------------------------------
//-----------------------------------------------------------------------------
// clear states on request
//-----------------------------------------------------------------------------
IF NOT Enable 
THEN
  _nCheckCount                := 0;
  _eState                     :=
  DetectMoverId               := E_XPU_CHECK.INIT_CHECK;
  RETURN;
END_IF
//-----------------------------------------------------------------------------
//-----------------------------------------------------------------------------
//  mover ID detection sequence
//-----------------------------------------------------------------------------
CASE _eState
OF
  E_XPU_CHECK.INIT_CHECK:
    IF Enable
    THEN
      IF NOT (_bInit)
      THEN
        _bInit                      := TRUE;

        _stMsg.eType                := E_MessageType.eMessageInfo;
        _stMsg.eSubdevice           := e_Subdevice.Xpu_fbProcessingUnit;
        _stMsg.iErrorNumber         := 0;
        _stMsg.sText                := concat('OperationMode', ': ');
        _stMsg.sText                := concat(_stMsg.sText, OpModeToString());
        f_MessageSet(_stMsg, _nXpu);

        _stMsg.eType                := E_MessageType.eMessageInfo;
        _stMsg.eSubdevice           := e_Subdevice.Xpu_fbProcessingUnit;
        _stMsg.iErrorNumber         := 0;
        _stMsg.sText                := concat(TO_STRING(E_XPU_CHECK.MOVER_ID_DETECTION_MODE), ': ');
        _stMsg.sText                := concat(_stMsg.sText, TO_STRING(IdDetectionModeToString()));
        f_MessageSet(_stMsg, _nXpu);
      END_IF

      _nCheckCount            := _nCheckCount + 1;
      IF (_nCheckCount MOD _nCheckModulo = 0)
      THEN
        _nCheckCount          := 0;
        _eState               := E_XPU_CHECK.MOVER_ID_DETECTION_MODE;
      END_IF
    END_IF
END_CASE
//-----------------------------------------------------------------------------
//-----------------------------------------------------------------------------
//  check for simulation or Standard ID detection
//-----------------------------------------------------------------------------
CASE _eState
OF
  E_XPU_CHECK.MOVER_ID_DETECTION_MODE:

    IF (_XpuOperationMode     = OperationMode.Simulation)
    THEN
      _eState                 := E_XPU_CHECK.INIT_CHECK;
      _eReturn                := E_XPU_CHECK.MOVER_ID_SIMULATION;

    ELSIF (_MoverIdDetectionMode = MoverIdDetectionMode.Standard)
    THEN
      _eState                 := E_XPU_CHECK.INIT_CHECK;
      _eReturn                := E_XPU_CHECK.MOVER_ID_STANDARD;

    ELSIF (_MoverIdDetectionMode = MoverIdDetectionMode.Mover1)
    THEN
      _eState                 := 
      _eReturn                := E_XPU_CHECK.MOVER_ID_DETECTION_VALID;

    ELSE
      _eReturn                := E_XPU_CHECK.MOVER_ID_MULTIPLE_NOT_SUPPORTED;
    END_IF
END_CASE
//-----------------------------------------------------------------------------
//-----------------------------------------------------------------------------
//
//-----------------------------------------------------------------------------
CASE _eState
OF
  //---------------------------------------------------------------------------
  E_XPU_CHECK.MOVER_ID_DETECTION_VALID:

    IF (_fbProcessingUnit.GetIsMoverIdDetectionValid())
    THEN
      IF NOT (_bMoverIdDetectionValid)
      THEN
        _stMsg.eType                := E_MessageType.eMessageInfo;
        _stMsg.eSubdevice           := e_Subdevice.Xpu_fbProcessingUnit;
        _stMsg.iErrorNumber         := 0;
        _stMsg.sText                := concat(TO_STRING(E_XPU_CHECK.MOVER_ID_DETECTION_VALID), ': ');
        _stMsg.sText                := concat(_stMsg.sText, TO_STRING(E_PROGRESS.PROGRESS_DONE));
        f_MessageSet(_stMsg, _nXpu);
      END_IF

      _bMoverIdDetectionValid := TRUE;

      _eReturn                := E_XPU_CHECK.MOVER_ID_DETECTION_VALID;
      _eState                 := E_XPU_CHECK.INIT_CHECK;
    ELSE
      _bMoverIdDetectionValid := FALSE;

      _eState                 := E_XPU_CHECK.MOVER_ID_DETECTION_DC_LINK;

      IF (_eMessageLevel = E_MessageType.eMessageVerbose)
      THEN
        _stMsg.eType          := E_MessageType.eMessageVerbose;
        _stMsg.eSubdevice     := e_Subdevice.Xpu_fbProcessingUnit;
        _stMsg.iErrorNumber   := 0;
        _stMsg.sText          := concat(TO_STRING(_eReturn), ': ');
        _stMsg.sText          := concat(_stMsg.sText, TO_STRING(_eState));
        f_MessageSet(_stMsg, _nXpu);
      END_IF
    END_IF

  //---------------------------------------------------------------------------
  E_XPU_CHECK.MOVER_ID_DETECTION_DC_LINK:
    _eReturn                  := E_XPU_CHECK.MOVER_ID_DETECTION_DC_LINK;

    IF AllModulesDcLink       // wait for DcLink on all motor modules
    THEN
      IF (_fbProcessingUnit.TriggerMoverIdDetection())
      THEN
        _eState               := E_XPU_CHECK.MOVER_ID_DETECTION_BUSY;

        IF (_eMessageLevel = E_MessageType.eMessageVerbose)
        THEN
          _stMsg.eType        := E_MessageType.eMessageVerbose;
          _stMsg.eSubdevice   := e_Subdevice.Xpu_fbProcessingUnit;
          _stMsg.iErrorNumber := 0;
          _stMsg.sText        := concat(TO_STRING(_eReturn), ': ');
          _stMsg.sText        := concat(_stMsg.sText, TO_STRING(_eState));
          f_MessageSet(_stMsg, _nXpu);
        END_IF
      END_IF
    END_IF

  //---------------------------------------------------------------------------
  E_XPU_CHECK.MOVER_ID_DETECTION_BUSY:
    _eReturn                  := E_XPU_CHECK.MOVER_ID_DETECTION_BUSY;

    IF (_fbProcessingUnit.GetIsMoverIdDetectionActive())
    THEN
      _eState                 := E_XPU_CHECK.MOVER_ID_DETECTION_IDLE;

      IF (_eMessageLevel = E_MessageType.eMessageVerbose)
      THEN
        _stMsg.eType          := E_MessageType.eMessageVerbose;
        _stMsg.eSubdevice     := e_Subdevice.Xpu_fbProcessingUnit;
        _stMsg.iErrorNumber   := 0;
        _stMsg.sText          := concat(TO_STRING(_eReturn), ': ');
        _stMsg.sText          := concat(_stMsg.sText, TO_STRING(_eState));
        f_MessageSet(_stMsg, _nXpu);
      END_IF
    END_IF
END_CASE
//-----------------------------------------------------------------------------
//-----------------------------------------------------------------------------
//
//-----------------------------------------------------------------------------
CASE _eState
OF
  E_XPU_CHECK.MOVER_ID_DETECTION_IDLE:
    _eReturn                  := E_XPU_CHECK.MOVER_ID_DETECTION_IDLE;

    IF NOT(_fbProcessingUnit.GetIsMoverIdDetectionActive())
    THEN
      _eState                 := E_XPU_CHECK.MOVER_ID_DETECTION_STATE;

      IF (_eMessageLevel = E_MessageType.eMessageVerbose)
      THEN
        _stMsg.eType          := E_MessageType.eMessageVerbose;
        _stMsg.eSubdevice     := e_Subdevice.Xpu_fbProcessingUnit;
        _stMsg.iErrorNumber   := 0;
        _stMsg.sText          := concat(TO_STRING(_eReturn), ': ');
        _stMsg.sText          := concat(_stMsg.sText, TO_STRING(_eState));
        f_MessageSet(_stMsg, _nXpu);
      END_IF
    END_IF

  //---------------------------------------------------------------------------
  E_XPU_CHECK.MOVER_ID_DETECTION_STATE:
    _eReturn                  := E_XPU_CHECK.MOVER_ID_DETECTION_STATE;

    IF NOT(_fbProcessingUnit.GetHasMoverIdDetectionError())
    THEN
      _bMoverIdDetectionError := FALSE;

      _eState                 := E_XPU_CHECK.MOVER_ID_DETECTION_MODE;

      IF (_eMessageLevel = E_MessageType.eMessageVerbose)
      THEN
        _stMsg.eType          := E_MessageType.eMessageVerbose;
        _stMsg.eSubdevice     := e_Subdevice.Xpu_fbProcessingUnit;
        _stMsg.iErrorNumber   := 0;
        _stMsg.sText          := concat(TO_STRING(_eReturn), ': ');
        _stMsg.sText          := concat(_stMsg.sText, TO_STRING(e_progress.PROGRESS_DONE));
        f_MessageSet(_stMsg, _nXpu);
      END_IF
    ELSE
      IF NOT (_bMoverIdDetectionError)
      THEN
        _stMsg.eType          := E_MessageType.eMessageError;
        _stMsg.eSubdevice     := e_Subdevice.Xpu_fbProcessingUnit;
        _stMsg.iErrorNumber   := 0;
        _stMsg.sText          := concat(TO_STRING(_eReturn), ': ');
        _stMsg.sText          := concat(_stMsg.sText, TO_STRING(e_progress.PROGRESS_ERROR));
        f_MessageSet(_stMsg, _nXpu);
      END_IF

      _bMoverIdDetectionValid := FALSE;
      _bMoverIdDetectionError := TRUE;
    END_IF
END_CASE
//-----------------------------------------------------------------------------
//-----------------------------------------------------------------------------
//
//-----------------------------------------------------------------------------
DetectMoverId                 := _eReturn;
//-----------------------------------------------------------------------------
//-----------------------------------------------------------------------------
END_METHOD

PROPERTY State : REFERENCE TO ST_XPU_STATE
SET
_State ref= State;
END_SET
END_PROPERTY

END_FUNCTION_BLOCK

// ---- XTS/Xpu/fb_Xpu.TcPOU
//---------------------------------------------------------------------------------------------------------------
//
//  HAUD 2023.12.14
//
//  - XTS_TRANSPORT_LAYER
//
//  fb_Xpu
//  - connect XTS_Utility.lib to TcCom
//  - cyclic plausibility checks
//  - cyclic ModuleInfoData
//
//  - connection to TcCom Server for local FB instances
//
//
//  CTRL / STATE --> see proprerties
//  structs for use of function block via mapping
//  cyclic check for new command
//
//  VAR INPUT / OUTPUT --> see properties
//
//---------------------------------------------------------------------------------------------------------------
// This SOFTWARE is provided as an Exemple by THE PROVIDER "as is" and "with all faults." THE PROVIDER makes no 
// representations or warranties of any kind concerning the safety, suitability, lack of viruses, inaccuracies, 
// typographical errors, or other harmful components of this SOFTWARE. There are inherent dangers in the use of 
// any software, and you are solely responsible for determining whether this SOFTWARE is compatible with your 
// equipment and other software installed on your equipment. You are also solely responsible for the protection 
// of your equipment and backup of your data, and THE PROVIDER will not be liable for any damages you may suffer 
// in connection with using, modifying, or distributing this SOFTWARE.
//---------------------------------------------------------------------------------------------------------------
FUNCTION_BLOCK fb_Xpu //IMPLEMENTS I_Xpu
VAR
  _eCheck                     : E_XPU_CHECK;
  _eInit                      : E_XPU_INIT;       // MUST equal INIT_DONE for anything to work
  _sVersionXpu                : STRING(80);       // only valid after successful init
  _sVersionNctController      : STRING(80);       // only valid afetr successful init
  //-------------------------------------------------------------------------------------------------
  // XTS Environment; ProcessingUnit, Part, Track, Mover
  //  - instances are initialized by getting OTCIDs
  //-------------------------------------------------------------------------------------------------
  _nXpu                       : UINT := 1;  // input property in case of multiple XPU in project
  _nGroup                     : UINT;       // input property in case of multiple Xpu in project

  _nTrack                     : UINT := 1;  // this example is intended for one track only

  {attribute 'displaymode':='hex'}
  _CaGroupOID                 : OTCID; // input property frome cyclic CA group interface, MUST be set in order to do successful INIT

  // checked and evaluated in XpuCheckCycle()
  _bAllPositionsValid,
  _bMoverIdDetectionValid,
  _bMoverIdDetectionError     : BOOL;

  _nDetectedMoverCount,
  _nExpectedMoverCount        : UINT;

  _XpuOperationMode           : OperationMode;
  _MoverIdDetectionMode       : MoverIdDetectionMode;

  // XTS_Utility connection to TcCOM Object
  _fbEnvironment              : Tc3_XTS_Utility.FB_TcIoXtsEnvironment;

  // local instances of members of Environment
  // local members are connected to TcCOM by XpuInit()
  _fbProcessingUnit           : Tc3_XTS_Utility.FB_TcIoXtsProcessingUnit;

  _fbXpuPart                  : Tc3_XTS_Utility.FB_TcIoXtsXpuPart;
  _fbXpuTrack                 : Tc3_XTS_Utility.FB_TcIoXtsXpuTrack;

  _fbMc2CaGroup               : Tc3_XTS_Utility.FB_Mc2CaGroup;

  _fbPartModules              : ARRAY[1..MAX_MODULE]  OF Tc3_XTS_Utility.FB_TcIoXtsPartModule;
  _fbMoverXpu                 : ARRAY[1..MAX_MOVER]   OF Tc3_XTS_Utility.FB_TcIoXtsXpuMover;

  _fbParameterSet             : ARRAY[1..MAX_PARAMETER_SET] OF Tc3_XTS_Utility.FB_TcIoXtsParameterSet;

  _fbNctController            : Tc3_XTS_Utility.FB_TcIoXtsNctController;

  _ItfNctBaseUnit              : ARRAY[1..MAX_NCT_BASE_UNIT] OF Tc3_XTS_Utility.I_TcIoXtsNctBaseUnitInterface;


  // TcCOM ObjectId (who am I talking to?)
  {attribute 'displaymode':='hex'}
  _Xpu_OTCID                  : OTCID;
  {attribute 'displaymode':='hex'}
  _Nct_OTCID                  : OTCID;
  {attribute 'displaymode':='hex'}
  _Group_OTCID                : ARRAY[1..MAX_GROUP]         OF OTCID; // OTCID read from XPU
  {attribute 'displaymode':='hex'}
  _Part_OTCID                 : ARRAY[1..MAX_PART]          OF OTCID;
  {attribute 'displaymode':='hex'}
  _Track_OTCID                : ARRAY[1..MAX_TRACK]         OF OTCID;
  {attribute 'displaymode':='hex'}
  _Mov_OTCID                  : ARRAY[1..MAX_MOVER]         OF OTCID;
  {attribute 'displaymode':='hex'}
  _Module_OTCID               : ARRAY[1..MAX_MODULE]        OF OTCID;
  {attribute 'displaymode':='hex'}
  _ParameterSet_OTCID         : ARRAY[1..MAX_PARAMETER_SET] OF OTCID;
  {attribute 'displaymode':='hex'}
  _NctBaseUnit_OTCID          : ARRAY[1..MAX_NCT_BASE_UNIT] OF OTCID;

  // COE Data access
  _ModuleInfoData             : REFERENCE TO ARRAY[1..MAX_MODULE] OF Tc3_XTS_Utility.ST_InfoDataView;
  _bModulePower               : ARRAY[1..MAX_MODULE] OF BOOL;

  // double check RailLength, XpuInit() will get stuck in error if not configured correctly
  _RailLengthXpu              : LREAL;
  _RailLengthGroup            : LREAL;

  _nLengthXpu,
  _nLengthGroup               : UINT;

  _nNctBaseUnitCount,
  _nParameterSetCount,
  _nInfoServerCount,
  _nIfoStationCount,
  _nPartCount,
  _nTrackCount,
  _nTaskCount,
  _nMoverCount,
  _nModuleCount               : UINT;

  _ix                         : UINT;

  {attribute 'hide'}
  _XpuInfo                    : ST_XPU_INFO;

  _stMsg                      : ST_Message;
  _eMessageLevel              : E_MessageType;
END_VAR

// get DcLink information from motor modules
PROPERTY AllModulesDcLink : bool
GET
VAR
  _bTmp     : BOOL;
  _nModule  : UINT;
END_VAR
IF NOT (_eInit = E_XPU_INIT.INIT_DONE) THEN RETURN; END_IF

FOR _nModule := 1 TO _nModuleCount
DO
  IF NOT _bModulePower[_nModule] // information comes from cyclic call in Cycle(): ModuleInfoData()
  THEN
    _bTmp  := FALSE;
    EXIT;
  ELSE
    _bTmp  := TRUE;
  END_IF
END_FOR

AllModulesDcLink := _bTmp;
END_GET
END_PROPERTY

PROPERTY CaGroupOID : OTCID
SET
// Group OTCID must come from the CA Group mapping in NC.Objects
_CaGroupOID := CaGroupOID;
END_SET
END_PROPERTY

METHOD Cycle : E_PROGRESS
VAR_INPUT
  Enable      : BOOL; // enable to do cyclic checks on Environment and its members
END_VAR
VAR_IN_OUT
  _eChk       : E_XPU_CHECK;
END_VAR
VAR_INST

  _eJobResult,
  _eResult      : E_PROGRESS;
  _eState       : E_PROGRESS := E_PROGRESS.PROGRESS_INIT;

END_VAR
IF NOT Enable
THEN
  ModuleInfoData(FALSE);

  _eResult  :=
  _eState   := E_PROGRESS.PROGRESS_INIT; 
  _eChk     := E_XPU_CHECK.INIT_CHECK;
END_IF 
//-----------------------------------------------------------------------------
// cyclic data fetch from Environment, ProcessingUnit, Part, ...
//-----------------------------------------------------------------------------
CASE _eState
OF
  E_PROGRESS.PROGRESS_INIT:
    IF Enable
    THEN
      _eState := _eResult         := E_PROGRESS.PROGRESS_BUSY;
    END_IF

  //---------------------------------------------------------------------------
  E_PROGRESS.PROGRESS_BUSY:       // get data from Xpu, ProcessingUnit, Part, XpuCaGroup
    _eState                       := E_PROGRESS.PROGRESS_STARTUP;

    _bAllPositionsValid           := _fbProcessingUnit.GetAreAllPositionsValid();
    _nDetectedMoverCount          := TO_UINT(_fbProcessingUnit.GetDetectedMoverCount());
    _nExpectedMoverCount          := TO_UINT(_fbProcessingUnit.GetExpectedMoverCount());
  
    _XpuOperationMode             := _fbProcessingUnit.GetOperationMode();
    _MoverIdDetectionMode         := _fbProcessingUnit.GetMoverIdDetectionMode();
  
    _RailLengthXpu                := _fbXpuPart.GetLength();
    _RailLengthGroup              := _fbMc2CaGroup.GetRailLength();
    _nLengthXpu                   := TO_UINT(_RailLengthXpu);
    _nLengthGroup                 := TO_UINT(_RailLengthGroup);
END_CASE
//-----------------------------------------------------------------------------
//-----------------------------------------------------------------------------
CASE _eState
OF
  //---------------------------------------------------------------------------
  E_PROGRESS.PROGRESS_STARTUP:    // check data for errors
    IF NOT (_bAllPositionsValid)
    THEN
      _eChk                       := E_XPU_CHECK.PROCESSING_UNIT_POSITIONS_VALID;
      _eState := _eResult         := E_PROGRESS.PROGRESS_ERROR;

      _stMsg.eType                := E_MessageType.eMessageError;
      _stMsg.eSubdevice           := e_Subdevice.Xpu_fbProcessingUnit;
      _stMsg.iErrorNumber         := 0;
      _stMsg.sText                := concat(TO_STRING(E_XPU_CHECK.PROCESSING_UNIT_POSITIONS_VALID), ': ');
      _stMsg.sText                := concat(_stMsg.sText, TO_STRING(_eResult));
      f_MessageSet(_stMsg, _nXpu);

    ELSIF NOT (_nLengthXpu > 0)
    THEN
      _eChk                       := E_XPU_CHECK.XPU_RAIL_LENGTH;
      _eState := _eResult         := E_PROGRESS.PROGRESS_ERROR;

      _stMsg.eType                := E_MessageType.eMessageError;
      _stMsg.eSubdevice           := e_Subdevice.Xpu_fbProcessingUnit;
      _stMsg.iErrorNumber         := 0;
      _stMsg.sText                := concat(TO_STRING(E_XPU_CHECK.XPU_RAIL_LENGTH), ': ');
      _stMsg.sText                := concat(_stMsg.sText, TO_STRING(_eResult));
      f_MessageSet(_stMsg, _nXpu);

    ELSIF NOT (_nLengthGroup > 0)
    THEN
      _eChk                       := E_XPU_CHECK.GROUP_RAIL_LENGTH;
      _eState := _eResult         := E_PROGRESS.PROGRESS_ERROR;
     
      _stMsg.eType                := E_MessageType.eMessageError;
      _stMsg.eSubdevice           := e_Subdevice.Xpu_fbProcessingUnit;
      _stMsg.iErrorNumber         := 0;
      _stMsg.sText                := concat(TO_STRING(E_XPU_CHECK.GROUP_RAIL_LENGTH), ': ');
      _stMsg.sText                := concat(_stMsg.sText, TO_STRING(_eResult));
      f_MessageSet(_stMsg, _nXpu);

    ELSIF NOT (_nDetectedMoverCount = _nExpectedMoverCount)
    THEN
      _bMoverIdDetectionValid     := FALSE;
      _eChk                       := E_XPU_CHECK.MOVER_COUNT_NOT_EQUAL;
      _eState := _eResult         := E_PROGRESS.PROGRESS_ERROR;

      _stMsg.eType                := E_MessageType.eMessageError;
      _stMsg.eSubdevice           := e_Subdevice.Xpu_fbProcessingUnit;
      _stMsg.iErrorNumber         := 0;
      _stMsg.sText                := concat(TO_STRING(E_XPU_CHECK.MOVER_COUNT_NOT_EQUAL), ': ');
      _stMsg.sText                := concat(_stMsg.sText, TO_STRING(_eResult));
      f_MessageSet(_stMsg, _nXpu);
  
    ELSIF NOT (_nLengthXpu = _nLengthGroup)
    THEN
      _eChk                       := E_XPU_CHECK.RAIL_LENGTH_COMPARE;
      _eState := _eResult         := E_PROGRESS.PROGRESS_ERROR;
 
      _stMsg.eType                := E_MessageType.eMessageError;
      _stMsg.eSubdevice           := e_Subdevice.Xpu_fbProcessingUnit;
      _stMsg.iErrorNumber         := 0;
      _stMsg.sText                := concat(TO_STRING(E_XPU_CHECK.RAIL_LENGTH_COMPARE), ': ');
      _stMsg.sText                := concat(_stMsg.sText, TO_STRING(_eResult));
      f_MessageSet(_stMsg, _nXpu);

    ELSE
      _eResult                    := E_PROGRESS.PROGRESS_WORKING;

      IF NOT (__ISVALIDREF(_ModuleInfoData))
      THEN
        _eState                   := E_PROGRESS.PROGRESS_BUSY;

        _stMsg.eType              := E_MessageType.eMessageError;
        _stMsg.eSubdevice         := e_Subdevice.Xpu_fbPartModules;
        _stMsg.iErrorNumber       := 0;
        _stMsg.sText              := concat(TO_STRING(_eState), ': ');
        _stMsg.sText              := concat(_stMsg.sText, 'NOT VALID _ModuleInfoData ref');
      ELSE
        _eJobResult               := ModuleInfoData(TRUE);
  
        IF (_eJobResult = E_PROGRESS.PROGRESS_DONE)
        THEN
          _eState                 := E_PROGRESS.PROGRESS_BUSY;
        END_IF  
      END_IF
    END_IF
END_CASE

Cycle                             := _eResult;
END_METHOD

METHOD GetEnvironment : I_TcIoXtsEnvironment
VAR_INPUT
END_VAR
IF NOT (_eInit = E_XPU_INIT.INIT_DONE) THEN RETURN; END_IF

GetEnvironment := _fbEnvironment;
END_METHOD

METHOD GetNctBaseUnit : Tc3_XTS_Utility.I_TcIoXtsNctBaseUnitInterface
VAR_INPUT
  Index     : UINT;
END_VAR
IF NOT (_eInit = E_XPU_INIT.INIT_DONE) THEN RETURN; END_IF

IF NOT (Index > 0) OR
   NOT (Index < MAX_NCT_BASE_UNIT+1)
THEN
  RETURN;
ELSE
  GetNctBaseUnit    := _ItfNctBaseUnit[Index];
END_IF
END_METHOD

METHOD GetNctController : Tc3_XTS_Utility.I_TcIoXtsNctController
VAR_INPUT
END_VAR
IF NOT (_eInit = E_XPU_INIT.INIT_DONE) THEN RETURN; END_IF

GetNctController := _fbNctController;
END_METHOD

METHOD GetParameterSet : I_TcIoXtsParameterSet
VAR_INPUT
  Index     : UINT;
END_VAR
IF NOT (_eInit = E_XPU_INIT.INIT_DONE) THEN RETURN; END_IF

IF NOT (Index > 0) OR
   NOT (Index < MAX_PARAMETER_SET+1)
THEN
  RETURN;
ELSE
  GetParameterSet   := _fbParameterSet[Index];
END_IF
END_METHOD

METHOD GetProcessingUnit : Tc3_XTS_Utility.I_TcIoXtsProcessingUnit
VAR_INPUT
END_VAR
IF NOT (_eInit = E_XPU_INIT.INIT_DONE) THEN RETURN; END_IF

GetProcessingUnit := _fbProcessingUnit;
END_METHOD

METHOD GetXpuMover : Tc3_XTS_Utility.I_TcIoXtsXpuMover
VAR_INPUT
  Index     : UINT;
END_VAR
IF NOT (_eInit = E_XPU_INIT.INIT_DONE) THEN RETURN; END_IF

IF NOT (Index > 0) OR
   NOT (Index < MAX_MOVER+1)
THEN
  RETURN;
ELSE
  GetXpuMover   := _fbMoverXpu[Index];
END_IF
END_METHOD

// mothers' little helper for display in visu
METHOD IdDetectionModeToString : string(20)
VAR
  _DetectionMode    : MoverIdDetectionMode; // Mover ID detection procedure
END_VAR
// just a little helper for visu display
IF NOT (_eInit = E_XPU_INIT.INIT_DONE) THEN IdDetectionModeToString := 'INIT required'; RETURN; END_IF

_DetectionMode := _fbProcessingUnit.GetMoverIdDetectionMode();

CASE _DetectionMode
OF
  MoverIdDetectionMode.Standard:
    IdDetectionModeToString       := 'Standard';

  MoverIdDetectionMode.Mover1:
    IdDetectionModeToString       := 'Mover 1';

  MoverIdDetectionMode.MultipleMover1:
    IdDetectionModeToString       := 'Multiple Mover 1';

ELSE
    IdDetectionModeToString       := 'UNKNOWN Mode';
END_CASE
END_METHOD

PROPERTY MessageLevel : e_messagetype
SET
_eMessageLevel := MessageLevel;
END_SET
END_PROPERTY

// mothers' little helper for display in visu
METHOD PRIVATE ModuleInfoData : E_PROGRESS
VAR_INPUT
  Enable        : BOOL; // enable to read ST_InfoDataView for diag/display
END_VAR
VAR_INST
  _idt,
  _nModule : UINT;
  _eReturn,
  _eState       : E_PROGRESS;
  _aPcbTemp     : ARRAY[1..4] OF REAL;
END_VAR
//---------------------------------------------------------------------------------------------
// just a little helper for visu display
// collects module data for local data
//---------------------------------------------------------------------------------------------
IF NOT (_eInit = E_XPU_INIT.INIT_DONE)      // if Xpu init is not done, just leave
THEN 
  RETURN; 
END_IF
//---------------------------------------------------------------------------------------------
IF NOT Enable                               // clear states on request
THEN
  _eReturn                                  := 
  _eState                                   := E_PROGRESS.PROGRESS_INIT; 
END_IF 
//---------------------------------------------------------------------------------------------
IF NOT (__ISVALIDREF(_ModuleInfoData))      // datafield not connected, error and leave
THEN
  ModuleInfoData                            := E_PROGRESS.PROGRESS_ERROR;
  RETURN;
END_IF
//---------------------------------------------------------------------------------------------
CASE _eState                                // get InfoData from motor modules
OF
  //-------------------------------------------------------------------------------------------
  E_PROGRESS.PROGRESS_INIT:
    IF Enable
    THEN
      _eState                                             := E_PROGRESS.PROGRESS_BUSY;
      _nModule                                            := 1;
    END_IF
END_CASE
CASE _eState
OF
  //-------------------------------------------------------------------------------------------
  E_PROGRESS.PROGRESS_BUSY:
    _eState                                               := E_PROGRESS.PROGRESS_PREPARE;

    _ModuleInfoData[_nModule].fAuxiliaryVoltage_5V        := _fbPartModules[_nModule].GetAuxiliaryVoltage5V();
    _ModuleInfoData[_nModule].fAuxiliaryVoltage_10V       := _fbPartModules[_nModule].GetAuxiliaryVoltage10V();
    _ModuleInfoData[_nModule].fAuxiliaryVoltage_24V       := _fbPartModules[_nModule].GetAuxiliaryVoltage24V();

    _ModuleInfoData[_nModule].fDcLinkVoltage              := _fbPartModules[_nModule].GetDCLinkVoltage();

    IF (_ModuleInfoData[_nModule].fDcLinkVoltage > 48.0*0.85) AND
       (_ModuleInfoData[_nModule].fDcLinkVoltage < 48.0*1.15)
    THEN
      _bModulePower[_nModule]                             := TRUE;
    ELSE
      _bModulePower[_nModule]                             := SEL((_XpuOperationMode = OperationMode.Simulation), FALSE, TRUE);
    END_IF

    _ModuleInfoData[_nModule].nCurrentScaling             := TO_INT(_fbPartModules[_nModule].GetCurrentScaling());

    _ModuleInfoData[_nModule].nDeviceInfo                 := _fbPartModules[_nModule].GetDeviceInfo();

    IF (_XpuOperationMode = OperationMode.Normal)
    THEN
      _ModuleInfoData[_nModule].fAverageTemp              := 0.0;
  
      _aPcbTemp                                           := _fbPartModules[_nModule].GetPCBTemperatures();
  
      _ModuleInfoData[_nModule].fPcbTemp_0                := _aPcbTemp[1];
      _ModuleInfoData[_nModule].fPcbTemp_1                := _aPcbTemp[2];
      _ModuleInfoData[_nModule].fPcbTemp_2                := _aPcbTemp[3];
      _ModuleInfoData[_nModule].fPcbTemp_3                := _aPcbTemp[4];

      FOR _idt := 1 TO 4
      DO
        _ModuleInfoData[_nModule].fAverageTemp            := _ModuleInfoData[_nModule].fAverageTemp + _aPcbTemp[_idt];
      END_FOR
      _ModuleInfoData[_nModule].fAverageTemp              := _ModuleInfoData[_nModule].fAverageTemp / 4;
    END_IF

    _ModuleInfoData[_nModule].fOverallCurrent             := _fbPartModules[_nModule].GetOverallCurrent();

    _ModuleInfoData[_nModule].fMaxDCLinkVoltageLast500ms  := _fbPartModules[_nModule].GetMaxDCLinkVoltageLast500ms();
    _ModuleInfoData[_nModule].fMaxOverallCurrentLast500ms := _fbPartModules[_nModule].GetMaxOverallCurrentLast500ms();
END_CASE
CASE _eState 
OF
  //-------------------------------------------------------------------------------------------
  E_PROGRESS.PROGRESS_PREPARE:
    IF (_nModule > _nModuleCount-1)
    THEN
      _eState                                             := E_PROGRESS.PROGRESS_WORKING;
    ELSE
      _nModule                                            := _nModule + 1;
      _eReturn                                            :=
      _eState                                             := E_PROGRESS.PROGRESS_BUSY;
    END_IF

  //-------------------------------------------------------------------------------------------
  E_PROGRESS.PROGRESS_WORKING:
    _eReturn                                              := E_PROGRESS.PROGRESS_DONE;
    _eState                                               := E_PROGRESS.PROGRESS_INIT;
END_CASE

ModuleInfoData                                            := _eReturn;
END_METHOD

// mothers' little helper for display in visu
METHOD MoverPositionAssignementToString : string(20)
VAR
  _PositionAssignement    : MoverPositionAssignment; // XPU movver assignement procedure
END_VAR
// just a little helper for visu display
IF NOT (_eInit = E_XPU_INIT.INIT_DONE) THEN MoverPositionAssignementToString := 'INIT required'; RETURN; END_IF

_PositionAssignement      := _fbProcessingUnit.GetMoverPositionAssignment();

CASE _PositionAssignement
OF
  MoverPositionAssignment.Standard:
    MoverPositionAssignementToString    := 'Standard';

  MoverPositionAssignment.StartAtFirstMover:
    MoverPositionAssignementToString    := 'Start At First Mover';
ELSE
    MoverPositionAssignementToString    := 'UNKNOWN Assgnement';
END_CASE
END_METHOD

// mothers' little helper for display in visu
METHOD OpModeToString : String(20)
VAR
  _OpMode     : OperationMode; // XPU operation mode
END_VAR
// just a little helper for visu display
IF NOT (_eInit = E_XPU_INIT.INIT_DONE) THEN OpModeToString := 'INIT required'; RETURN; END_IF

_OpMode   := _fbProcessingUnit.GetOperationMode();

CASE _OpMode
OF
  OperationMode.Normal:
    OpModeToString      := 'Normal';

  OperationMode.Simulation:
    OpModeToString      := 'Simulation';

ELSE
    OpModeToString      := 'UNKNOWN OP MODE';
END_CASE
END_METHOD

PROPERTY RailLength : lreal
GET
IF (_eInit = E_XPU_INIT.INIT_DONE)
THEN
  RailLength := _fbXpuPart.GetLength();
ELSE
  RailLength := 0.0;
END_IF
END_GET
END_PROPERTY

PROPERTY XpuInfo : st_xpu_info
GET
IF NOT (_eInit = E_XPU_INIT.INIT_DONE) THEN RETURN; END_IF

_XpuInfo.AllPositionsValid        := _bAllPositionsValid;

_XpuInfo.IdDetectionError         := _bMoverIdDetectionError;
_XpuInfo.IdDetectionValid         := _bMoverIdDetectionValid;

_XpuInfo.IdDetectionActive        := _fbProcessingUnit.GetIsMoverIdDetectionActive();

_XpuInfo.OperationMode            := TO_UINT(_fbProcessingUnit.GetOperationMode());

_XpuInfo.IdDetectionMode          := TO_UINT(_fbProcessingUnit.GetMoverIdDetectionMode());
_XpuInfo.MoverPositionAssignement := TO_UINT(_fbProcessingUnit.GetMoverPositionAssignment());

_XpuInfo.nDetectedAxisCount       := _nDetectedMoverCount;
_XpuInfo.nExpectedAxisCount       := _nExpectedMoverCount;

_XpuInfo.nParameterSetCount       := _nParameterSetCount;

XpuInfo := _XpuInfo;
END_GET
END_PROPERTY

METHOD PROTECTED XpuInit  : E_XPU_INIT      // connect to TcCOM
VAR_INPUT
  Execute       : BOOL;           // must be executed for connecting to TcCOM Environment of Xpu
END_VAR
VAR_IN_OUT
  _eReslt       : E_PROGRESS;     // send info about progress to caller
  _eChk         : E_XPU_CHECK;
END_VAR
VAR_INST
  _eState           : E_PROGRESS;   // progress state
  _nState           : E_XPU_INIT;   // initialization state
  _eDataGetCount    : E_PROGRESS;   // cycle counter to catch exceeding wait time for data from ProcessingUnit

  _nParaSetIdx      : UINT;

  _nMoverIdx,
  _nModuleIdx       : UINT;

  _nNctBaseUnitIdx        : UINT;
END_VAR
//-----------------------------------------------------------------------------------------------
//-----------------------------------------------------------------------------------------------
// clear progress on request
IF NOT Execute 
THEN 
  _eState                           := E_PROGRESS.PROGRESS_INIT;
  _eDataGetCount                    := 0;
 
  XpuInit                           :=
  _nState                           := E_XPU_INIT.INIT_START; 
  RETURN; 
END_IF
//-----------------------------------------------------------------------------------------------
//-----------------------------------------------------------------------------------------------
// progress state
//-----------------------------------------------------------------------------------------------
//-----------------------------------------------------------------------------------------------
CASE _eState
OF
  E_PROGRESS.PROGRESS_INIT:         // clear start
    IF Execute
    THEN
      _eState                       := E_PROGRESS.PROGRESS_BUSY;
      _eChk                         := E_XPU_CHECK.INIT_CHECK;    // clear cyclic check state
      _sVersionNctController        :=
      _sVersionXpu                  := TO_STRING(_eChk);          // clear Version string

      // always initialize environment function blocks to get defined start of progress
      _fbEnvironment.Init(FALSE);
      _fbEnvironment.GetXpuOids(FALSE);
      _fbEnvironment.GetInfoServerOids(FALSE);

      // clear initialization states
      _nState                       := E_XPU_INIT.INIT_START;

      // clear check bits
      _bAllPositionsValid           :=
      _bMoverIdDetectionValid       :=
      _bMoverIdDetectionError       := FALSE;

      // clear check values
      _nLengthXpu                   :=
      _nLengthGroup                 :=
      _nDetectedMoverCount          :=
      _nExpectedMoverCount          := 0;

      // clear work values
      _nNctBaseUnitCount            :=
      _nNctBaseUnitIdx              :=
      _nParameterSetCount           :=
      _nInfoServerCount             :=
      _nIfoStationCount             :=
      _nPartCount                   :=
      _nTrackCount                  :=
      _nTaskCount                   :=
      _nMoverCount                  :=
      _nModuleCount                 :=
      _nMoverIdx                    :=
      _nModuleIdx                   := 0;

      IF (_eMessageLevel = E_MessageType.eMessageVerbose)
      THEN
        _stMsg.eType                := E_MessageType.eMessageVerbose;
        _stMsg.eSubdevice           := e_Subdevice.Xpu_fbEnvironment;
        _stMsg.iErrorNumber         := 0;
        _stMsg.sText                := concat(TO_STRING(_eState), ': ');
        _stMsg.sText                := concat(_stMsg.sText, TO_STRING(_eChk));
        f_MessageSet(_stMsg, _nXpu);
      END_IF
    END_IF
END_CASE
//-----------------------------------------------------------------------------------------------
//-----------------------------------------------------------------------------------------------
//-----------------------------------------------------------------------------------------------
CASE _eState
OF
  E_PROGRESS.PROGRESS_BUSY:         // begin with initializing environment
    CASE _nState
    OF
  //-----------------------------------------------------------------------------------------------
  //-----------------------------------------------------------------------------------------------
  INIT_START:                       // call initialization of environment

    IF NOT _fbEnvironment.P_IsInitialized
    THEN
      _fbEnvironment.Init(TRUE);
    END_IF

    IF (_fbEnvironment.bError)
    THEN
      _eChk                         := E_XPU_CHECK.INIT_CHECK_ERROR;
                                    
      _stMsg.eType                  := E_MessageType.eMessageError;
      _stMsg.eSubdevice             := e_Subdevice.Xpu_fbEnvironment;
      _stMsg.iErrorNumber           := 666;
      _stMsg.sText                  := concat(TO_STRING(_eState), ': ');
      _stMsg.sText                  := concat(_stMsg.sText, TO_STRING(_eChk));
      f_MessageSet(_stMsg, _nXpu);

      _eState                       := E_PROGRESS.PROGRESS_ERROR;

    // get information about success in Property (P_<function>)
    ELSIF _fbEnvironment.P_IsInitialized
    THEN
      // now environment is initialized
     
      //---------------------------------------------------------------------
      // use of local function block instances
      // get information about Object IDs to local datafields
      //---------------------------------------------------------------------
      //  - everything else in this state machine is for use within fb_Xpu
      //  - the following states shall illustrate how TcCOM Objects are connected through XTS_Utility lib
      //  - local instances of members of Environment are connected from here onward
      //
      IF _fbEnvironment.GetXpuOids(TRUE) // get object IDs for all processing units
      THEN
        _fbEnvironment.Init(FALSE);// clear environment init
        _nState                     := INIT_ENVIRONMENT_OID;

        IF (_eMessageLevel = E_MessageType.eMessageVerbose)
        THEN
          _stMsg.eType              := E_MessageType.eMessageVerbose;
          _stMsg.eSubdevice         := e_Subdevice.Xpu_fbEnvironment;
          _stMsg.iErrorNumber       := 0;
          _stMsg.sText              := concat(TO_STRING(_eState), ': ');
          _stMsg.sText              := concat(_stMsg.sText, TO_STRING(_nState));
          f_MessageSet(_stMsg, _nXpu);
        END_IF
      END_IF
    END_IF

  //-----------------------------------------------------------------------------------------------
  //-----------------------------------------------------------------------------------------------
  INIT_ENVIRONMENT_OID:             // get processing unit object ID for THIS instance
    _Xpu_OTCID                      := _fbEnvironment.P_XpuOids[_nXpu];   // fb_Xpu.XpuInstance --> _nXpu

    // clear all local object IDs
    memset(ADR(_Part_OTCID)         , 0, SIZEOF(_Part_OTCID));
    memset(ADR(_Track_OTCID)        , 0, SIZEOF(_Track_OTCID));
    memset(ADR(_Mov_OTCID)          , 0, SIZEOF(_Mov_OTCID));
    memset(ADR(_Module_OTCID)       , 0, SIZEOF(_Module_OTCID));
    memset(ADR(_ParameterSet_OTCID) , 0, SIZEOF(_ParameterSet_OTCID));

    // clear function blocks
    _fbEnvironment.GetXpuOids           (FALSE);
    _fbEnvironment.GetCaGroupCount      (FALSE);
    _fbEnvironment.GetInfoServerCount   (FALSE);
    _fbEnvironment.GetParameterSetCount (FALSE);

    _eState                         := E_PROGRESS.PROGRESS_PREPARE; // TODO - implement InfoServer R/W
    _nState                         := INIT_CA_GROUP_OID;           // TODO - implement initialization states for info server procedure

    //_nState                       := INIT_INFO_SERVER_ITF;              // check environment for info servers

  //-----------------------------------------------------------------------------------------------
  //-----------------------------------------------------------------------------------------------
  INIT_INFO_SERVER_ITF:           // HAUD 2024 03 14: TODO - implement procedure for getting Info server data to local datafields
    IF _fbEnvironment.GetInfoServerCount(TRUE)
    THEN
      // how many of you are there?
      _nInfoServerCount             := _fbEnvironment.P_InfoServerCount;

      IF (_nInfoServerCount > 0)
      THEN
        // go do something with the data
        //
        //  TODO - get station coordinates
        _eState                     := E_PROGRESS.PROGRESS_PREPARE; // TODO - implement InfoServer R/W
        _nState                     := INIT_CA_GROUP_OID;           // TODO - implement initialization states for info server procedure

        IF (_eMessageLevel = E_MessageType.eMessageVerbose)
        THEN
          _stMsg.eType              := E_MessageType.eMessageVerbose;
          _stMsg.eSubdevice         := e_Subdevice.Xpu_fbEnvironment;
          _stMsg.iErrorNumber       := 0;
          _stMsg.sText              := concat(TO_STRING(_eState), ': ');
          _stMsg.sText              := concat(_stMsg.sText, TO_STRING(_nState));
          f_MessageSet(_stMsg, _nXpu);
        END_IF

      ELSE
        // no info server present
        _eState                     := E_PROGRESS.PROGRESS_PREPARE;
        _nState                     := INIT_CA_GROUP_OID; // go check CA group

        IF (_eMessageLevel = E_MessageType.eMessageVerbose)
        THEN
          _stMsg.eType              := E_MessageType.eMessageVerbose;
          _stMsg.eSubdevice         := e_Subdevice.Xpu_fbEnvironment;
          _stMsg.iErrorNumber       := 0;
          _stMsg.sText              := concat(TO_STRING(_eState), ': ');
          _stMsg.sText              := concat(_stMsg.sText, TO_STRING(_nState));
          f_MessageSet(_stMsg, _nXpu);
        END_IF
      END_IF
    END_IF
  END_CASE
END_CASE
//-----------------------------------------------------------------------------------------------
//-----------------------------------------------------------------------------------------------
//-----------------------------------------------------------------------------------------------
CASE _eState
OF
  E_PROGRESS.PROGRESS_PREPARE:      // CA group initialization
  CASE _nState
  OF
  //-----------------------------------------------------------------------------------------------
  //-----------------------------------------------------------------------------------------------
  INIT_CA_GROUP_OID:                // get object IDs of all CA groups in environment
    IF _fbEnvironment.GetCaGroupOids(TRUE)
    THEN
      _Group_OTCID                  := _fbEnvironment.P_CaGroupOids;  // copy all Ids to local
      _nState                       := INIT_CA_GROUP_GET_OID;

      IF (_eMessageLevel = E_MessageType.eMessageVerbose)
      THEN
        _stMsg.eType                := E_MessageType.eMessageVerbose;
        _stMsg.eSubdevice           := e_Subdevice.Xpu_fbEnvironment;
        _stMsg.iErrorNumber         := 0;
        _stMsg.sText                := concat(TO_STRING(_eState), ': ');
        _stMsg.sText                := concat(_stMsg.sText, TO_STRING(_nState));
        f_MessageSet(_stMsg, _nXpu);
      END_IF
    END_IF

  //-----------------------------------------------------------------------------------------------
  //-----------------------------------------------------------------------------------------------
  INIT_CA_GROUP_GET_OID:            // look for any CA group
    _fbEnvironment.GetCaGroupOids(FALSE);
    IF NOT (_Group_OTCID[1] <> 0)
    THEN
      // no group is configured in project --> error, go add/link CA Group in NC objects
      _eChk                         := E_XPU_CHECK.GROUP_NOT_CONFIGURED;
      _eState                       := E_PROGRESS.PROGRESS_ERROR;

      _stMsg.eType                  := E_MessageType.eMessageError;
      _stMsg.eSubdevice             := e_Subdevice.Xpu_fbEnvironment;
      _stMsg.iErrorNumber           := 0;
      _stMsg.sText                  := concat(TO_STRING(_eState), ': ');
      _stMsg.sText                  := concat(_stMsg.sText, TO_STRING(_nState));
      f_MessageSet(_stMsg, _nXpu);
    ELSE
      _nState                       := INIT_CA_GROUP_CHECK_OID; // get matching CA group

      IF (_eMessageLevel = E_MessageType.eMessageVerbose)
      THEN
        _stMsg.eType                := E_MessageType.eMessageVerbose;
        _stMsg.eSubdevice           := e_Subdevice.Xpu_fbEnvironment;
        _stMsg.iErrorNumber         := 0;
        _stMsg.sText                := concat(TO_STRING(_eState), ': ');
        _stMsg.sText                := concat(_stMsg.sText, TO_STRING(_nState));
        //f_MessageSet(_stMsg, _nXpu);
      END_IF
    END_IF

  //-----------------------------------------------------------------------------------------------
  //-----------------------------------------------------------------------------------------------
  INIT_CA_GROUP_CHECK_OID:          // ID must be found, there is one chance
    _eChk                           := E_XPU_CHECK.GROUP_OID_MISMATCH;
    _eState                         := E_PROGRESS.PROGRESS_ERROR;

    FOR _ix := 1 TO MAX_GROUP
    DO
      IF (_fbEnvironment.P_CaGroupOids[_ix] <> 0)
      THEN
        // check whether the input from cyclic interface can be found in XPU data
        IF (_fbEnvironment.P_CaGroupOids[_ix] = _CaGroupOID)  // _CaGroupOID must be linked from NC Objects into PLC (GROUP_REF)
        THEN

          _eState                   := E_PROGRESS.PROGRESS_PREPARE; // stay here
          _eChk                     := E_XPU_CHECK.INIT_CHECK;

          _nGroup                   := _ix;

          _fbEnvironment.GetCaGroupOids(FALSE);
          _nState                   := INIT_CA_GROUP_COM; // only continue if match was found

          IF (_eMessageLevel = E_MessageType.eMessageVerbose)
          THEN
            _stMsg.eType            := E_MessageType.eMessageVerbose;
            _stMsg.eSubdevice       := e_Subdevice.Xpu_fbEnvironment;
            _stMsg.iErrorNumber     := _CaGroupOID;
            _stMsg.sText            := concat(TO_STRING(_eState), ': ');
            _stMsg.sText            := concat(_stMsg.sText, TO_STRING(_nState));
            f_MessageSet(_stMsg, _nXpu);
          END_IF
          EXIT;
        END_IF
      END_IF
    END_FOR

    IF (_eState = E_PROGRESS.PROGRESS_ERROR)
    THEN
      _stMsg.eType                  := E_MessageType.eMessageError;
      _stMsg.eSubdevice             := e_Subdevice.Xpu_fbEnvironment;
      _stMsg.iErrorNumber           := _nGroup;
      _stMsg.sText                  := concat(TO_STRING(_eState), ': ');
      _stMsg.sText                  := concat(_stMsg.sText, TO_STRING(_nState));
      f_MessageSet(_stMsg, _nXpu);
    END_IF

  //-----------------------------------------------------------------------------------------------
  //-----------------------------------------------------------------------------------------------
  INIT_CA_GROUP_COM:                // connect to CaGroup function block in environment
    IF (_fbMc2CaGroup.GetComObject(_fbEnvironment.P_CaGroupOids[_nGroup]))
    THEN
      _fbEnvironment.GetParameterSetCount(FALSE);

      _nState                       := INIT_PARAMETERSET_COUNT;

      IF (_eMessageLevel = E_MessageType.eMessageVerbose)
      THEN
        _stMsg.eType                := E_MessageType.eMessageVerbose;
        _stMsg.eSubdevice           := e_Subdevice.Xpu_fbEnvironment;
        _stMsg.iErrorNumber         := _nGroup;
        _stMsg.sText                := concat(TO_STRING(_eState), ': ');
        _stMsg.sText                := concat(_stMsg.sText, TO_STRING(_nState));
       f_MessageSet(_stMsg, _nXpu);
      END_IF
    END_IF

